			iStartInstID := iStartInstID +1;
			iStartLED := 	iStartLED +1;
			
			Q_sConvString:=	CONCAT(Q_sConvString,F_ToCHR(I_sStartZeichen));
			Q_sConvString:=	CONCAT(Q_sConvString,DINT_TO_STRING(I_diID));
			Q_sConvString:=	CONCAT(Q_sConvString,'.LED.');
			Q_sConvString:=	CONCAT(Q_sConvString,INT_TO_STRING(iStartInstID));
			Q_sConvString:=	CONCAT(Q_sConvString,'.ON.');
			Q_sConvString:=	CONCAT(Q_sConvString,INT_TO_STRING(I_iLED[iStartLED]));
			Q_sConvString:=	CONCAT(Q_sConvString,F_ToCHR(I_sEndZeichen));
		ELSE
			(* Externe LEDs*)
			iStartInstIDExt := 65;
			iStartLEDExt := 1;
			
			Q_sConvString:=	CONCAT(F_ToCHR(I_sStartZeichen),DINT_TO_STRING(I_diID));
			Q_sConvString:=	CONCAT(Q_sConvString,'.LED.');
			Q_sConvString:=	CONCAT(Q_sConvString,INT_TO_STRING(iStartInstIDExt));
			Q_sConvString:=	CONCAT(Q_sConvString,'.ON.');
			Q_sConvString:=	CONCAT(Q_sConvString,INT_TO_STRING(I_iLEDExt[iStartLEDExt]));
			Q_sConvString:=	CONCAT(Q_sConvString,F_ToCHR(I_sEndZeichen));
			
			iStartInstIDExt := iStartInstIDExt +1;
			iStartLEDExt := 	iStartLEDExt +1;
			
			Q_sConvString:=	CONCAT(Q_sConvString,F_ToCHR(I_sStartZeichen));
			Q_sConvString:=	CONCAT(Q_sConvString,DINT_TO_STRING(I_diID));
			Q_sConvString:=	CONCAT(Q_sConvString,'.LED.');
			Q_sConvString:=	CONCAT(Q_sConvString,INT_TO_STRING(iStartInstIDExt));
			Q_sConvString:=	CONCAT(Q_sConvString,'.ON.');
			Q_sConvString:=	CONCAT(Q_sConvString,INT_TO_STRING(I_iLEDExt[iStartLEDExt]));
			Q_sConvString:=	CONCAT(Q_sConvString,F_ToCHR(I_sEndZeichen));
			
			iStartInstIDExt := iStartInstIDExt +1;
			iStartLEDExt := 	iStartLEDExt +1;
			
			Q_sConvString:=	CONCAT(Q_sConvString,F_ToCHR(I_sStartZeichen));
			Q_sConvString:=	CONCAT(Q_sConvString,DINT_TO_STRING(I_diID));
			Q_sConvString:=	CONCAT(Q_sConvString,'.LED.');
			Q_sConvString:=	CONCAT(Q_sConvString,INT_TO_STRING(iStartInstIDExt));
			Q_sConvString:=	CONCAT(Q_sConvString,'.ON.');
			Q_sConvString:=	CONCAT(Q_sConvString,INT_TO_STRING(I_iLEDExt[iStartLEDExt]));
			Q_sConvString:=	CONCAT(Q_sConvString,F_ToCHR(I_sEndZeichen));
			
			iStartInstIDExt := iStartInstIDExt +1;
			iStartLEDExt := 	iStartLEDExt +1;
			
			Q_sConvString:=	CONCAT(Q_sConvString,F_ToCHR(I_sStartZeichen));
			Q_sConvString:=	CONCAT(Q_sConvString,DINT_TO_STRING(I_diID));
			Q_sConvString:=	CONCAT(Q_sConvString,'.LED.');
			Q_sConvString:=	CONCAT(Q_sConvString,INT_TO_STRING(iStartInstIDExt));
			Q_sConvString:=	CONCAT(Q_sConvString,'.ON.');
			Q_sConvString:=	CONCAT(Q_sConvString,INT_TO_STRING(I_iLEDExt[iStartLEDExt]));
			Q_sConvString:=	CONCAT(Q_sConvString,F_ToCHR(I_sEndZeichen));
			
			iStartInstIDExt := iStartInstIDExt +1;
			iStartLEDExt := 	iStartLEDExt +1;
			
			Q_sConvString:=	CONCAT(Q_sConvString,F_ToCHR(I_sStartZeichen));
			Q_sConvString:=	CONCAT(Q_sConvString,DINT_TO_STRING(I_diID));
			Q_sConvString:=	CONCAT(Q_sConvString,'.LED.');
			Q_sConvString:=	CONCAT(Q_sConvString,INT_TO_STRING(iStartInstIDExt));
			Q_sConvString:=	CONCAT(Q_sConvString,'.ON.');
			Q_sConvString:=	CONCAT(Q_sConvString,INT_TO_STRING(I_iLEDExt[iStartLEDExt]));
			Q_sConvString:=	CONCAT(Q_sConvString,F_ToCHR(I_sEndZeichen));
			
			iStartInstIDExt := iStartInstIDExt +1;
			iStartLEDExt := 	iStartLEDExt +1;
			
			Q_sConvString:=	CONCAT(Q_sConvString,F_ToCHR(I_sStartZeichen));
			Q_sConvString:=	CONCAT(Q_sConvString,DINT_TO_STRING(I_diID));
			Q_sConvString:=	CONCAT(Q_sConvString,'.LED.');
			Q_sConvString:=	CONCAT(Q_sConvString,INT_TO_STRING(iStartInstIDExt));
			Q_sConvString:=	CONCAT(Q_sConvString,'.ON.');
			Q_sConvString:=	CONCAT(Q_sConvString,INT_TO_STRING(I_iLEDExt[iStartLEDExt]));
			Q_sConvString:=	CONCAT(Q_sConvString,F_ToCHR(I_sEndZeichen));
		END_IF
	END_IF
ELSE
	(* Reset *)
	Q_sConvString:=	CONCAT(F_ToCHR(I_sStartZeichen),DINT_TO_STRING(I_diID));
	Q_sConvString:=	CONCAT(Q_sConvString,'.SYS.');
	Q_sConvString:=	CONCAT(Q_sConvString,INT_TO_STRING(1));
	Q_sConvString:=	CONCAT(Q_sConvString,'.RESET');
	Q_sConvString:=	CONCAT(Q_sConvString,F_ToCHR(I_sEndZeichen));
END_IF

END_FUNCTION_BLOCK

// ---- POUs/RS485_Hausbus_FB/RS485 COM/fb_RS485Ping.TcPOU
(*======================================================================================================================================*)
(*fb_RS485Ping:	Einfacher Universal Ping Baustein um von allerlei Geräten von haus-bus.de Kommunikation zu Checken über RS485 
				im gegensatz zum ComCheck Baustein wird hier nur gelesen, da es Geräte gibt, welche entweder Zyklich selbst 
				ein Lebenszeichen geben z.B. CYD oder die 6Fach Taster (Helligkeit, Temp, Luftfeuchtigkeit).
				Besonderheit bei dem 6Fach Taster ist: nach einem Reset werden immer auch StatusTelegramme gesendet. 
				Damit lässt sich dann auch festellen ob ein Taster Online ist. 
				Für die Aktoren ist dieser Baustein eher weniger geeignet, da es dort keine Zyklischen Telegramme gibt und 
				auch nach einem Reset keine Statustelegramme gesendet werden! 
				
				Der Baustein kann auch verwendet werden um einfach nur zu überwachen, ob ein Teilnehmer noch online ist über langen
				Zeitraum- Dafür muss der Timeout einfach sehr Hoch gestellt werden - z.B 120 Minuten und bAutoPing Aktiviert sein 
			
				Wenn I_bAutoPing nicht Aktiv ist, wird nur eine Ping überprüfung beim Aktivieren des Bausteins über I_bExecute 
				durchgeführt. Wenn die Prüfung erfolgreich ist, wird der Status Q_bComOk gesetzt. Der Status Q_bComOk wird erst durch 
				I_bReset wieder zurück gesetzt. 
				
				Wenn I_bAutoPing Aktiv ist, wird sobald der Baustein über I_bExecute gestartet wurde, und ein Ping Aufgebaut ist, 
				immer nach ablauf der Zeit: I_tPingTimeout erneut der Ping geprüft. Sollte der Ping nicht kommen, so wird nach ablauf der 
+				Zeit: I_tPingTimeout in den Timepout gesprungen. Dann kann nur über einen Reset durch: I_bReset erneut gestartet werden*)
(*
Date          	| Version    	| created under        	| Author          	| Remark *)
(*====================================================================================================================================================*)
(*27/05/2025   	| 1.00      		| TC3		  		| N.Kersting       | first release *)
(*====================================================================================================================================================*)
FUNCTION_BLOCK fb_RS485Ping
VAR_INPUT
	I_bExecute			:BOOL;							(* Aktiviert den Ablauf *)
	I_bAutoPing			:BOOL;							(* Aktiviert die Automatische Prüfung, wenn aus- wird nur einmal beim Aktivieren über bExecute geprüft *)
	I_bAutoReset		:BOOL;							(* Aktiviert das Automatische wieder Quittieren wenn der Ping nicht empfangen wurde *)
	I_bReset			:BOOL;							(* Setzet den Ping und die Ablauf zurück *)
	I_tPingTimeout		:TIME := T#2S;					(* Zeit, bis der Ping gekommen sein muss *)
	I_diID				:DINT;							(* Device ID *)
	I_sStartZeichen		:BYTE := 16#FD;					(* Startzeichen Präfix *)
	I_sEndZeichen		:BYTE := 16#FE;					(* Endzeichen Suffix *)
	I_StringReceived	:STRING(255);					(* Empfangener String *)
END_VAR
VAR_OUTPUT		
	Q_sState			:STRING;						(* Status  *)
	Q_bComOk			:BOOL;							(* Verbindung Aufgebaut *)
	Q_bTimeout			:BOOL;							(* Timeout  *)
END_VAR
VAR
	bResetCnt			:BOOL;
	tonTimeout			:ton;
	icntSymbole			:INT;
	iStep				:INT;
	i					:INT;
	fbBusPingEvent		:fb_BusPingEvent;
	bCOMMem				:BOOL;
	rTrigFailCount		:r_trig;
	
	dwCntFail			:DWORD;
END_VAR

(* Timeout Zeit *)
tonTimeout(
	PT:= I_tPingTimeout);

(* Ping Fehler Zählen *)	
rTrigFailCount();
	
(* Reset ausführen *)
IF I_bReset 
	OR NOT I_bExecute
THEN
	iStep := 0;	
END_IF

(* Timeout Counter auf 0 Setzen *)
IF bResetCnt
THEN
	dwCntFail := 0;
END_IF
	
(* Ablauf *)
CASE iStep OF
(*=========================================================*)	
0:	Q_sState := 'INIT';
	Q_bComOk := FALSE;
	bCOMMem := FALSE; (* Ping zurück setzen *)
	tonTimeout.IN := FALSE;
	Q_bTimeout := FALSE;
	rTrigFailCount.CLK := FALSE;
	
	IF I_bExecute
	THEN
		iStep := iStep +1;
	END_IF
	
(*=========================================================*)	
1:	Q_sState :=  'Warten auf Ping ';	
	tonTimeout.IN := TRUE;
	
	IF fbBusPingEvent.Q_bOut
	THEN
		tonTimeout.IN := FALSE;
		bCOMMem := TRUE;
		iStep := 998;
	ELSIF
		tonTimeout.Q
	THEN
		tonTimeout.IN := FALSE;
		Q_bTimeout := TRUE;
		Q_bComOk := FALSE;
		Q_sState :=  'Timeout- Kein Ping empfangen';	
		iStep := -1;
	END_IF

(*=========================================================*)	
998: Q_sState :=  'Ping empfangen, Warte das String Leer ist';	
	tonTimeout.IN := TRUE;
	
	IF NOT fbBusPingEvent.Q_bOut
	THEN
		iStep := 999;
	ELSIF
		tonTimeout.Q
	THEN
		tonTimeout.IN := FALSE;
		Q_bTimeout := TRUE;
		Q_bComOk := FALSE;
		Q_sState :=  'Timeout String wurde nicht geleert!';	
		iStep := -998;
	END_IF
	
(*=========================================================*)	
999: Q_sState :=  'Ping empfangen, erfolgreich Verbunden!';		
	Q_bComOk := TRUE;
	Q_bTimeout := FALSE;
	
	(* Die Verbindung wurde nun geprüft, kann aber nur über
		I_bReset wieder erneut geprüft werden ! *)
	
	IF I_bAutoPing
	THEN
		tonTimeout.IN := TRUE;
		
		IF tonTimeout.Q
		THEN
			tonTimeout.IN := FALSE;
				
			IF I_bExecute
			THEN
				iStep := 1;	(* Erneut Prüfen *)
			END_IF
		END_IF
	ELSE
		tonTimeout.IN := FALSE;
	END_IF
ELSE
(*=========================================================*)	
(*	Timeout *)	
	rTrigFailCount.CLK := TRUE;
	
	IF rTrigFailCount.Q
	THEN
		dwCntFail := dwCntFail+1;
	END_IF
	(*	Automatische Quittierung *)	
	IF 	I_bAutoReset
	THEN
		tonTimeout.IN := TRUE;
		
		IF tonTimeout.Q
			OR fbBusPingEvent.Q_bOut
		THEN
			tonTimeout.IN := FALSE;
			
			IF I_bExecute
			THEN
				rTrigFailCount.CLK := FALSE;
				iStep := 1;	(* Erneut Prüfen *)
			END_IF
		END_IF
	END_IF
END_CASE


(* Durchgehend Checken ob Ping kommt *)
fbBusPingEvent(
	I_bReset := 			FALSE,
	I_sID:= 				DINT_TO_STRING(I_diID ), 
	I_sReceivedString:= 	I_StringReceived, 
	Q_bOut=> 				);

END_FUNCTION_BLOCK

// ---- POUs/RS485_Hausbus_FB/RelaisModul/fb_RelaisBus16F.TcPOU
(*======================================================================================================================================*)
(*fb_RelaisBus16F:		Einfache RS485 Kommunikation für Haus-bus.de Komponenten zum testen 	
						 *)
(*
Date          	| Version    	| created under        	| Author          	| Remark *)
(*====================================================================================================================================================*)
(*08/05/2025   	| 1.00      		| TC3		  		| N.Kersting       	| first release *)
(*08/05/2025   	| 1.01      		| TC3		  		| N.Kersting       	| Relais in Sections aufgeteilt um String Länge zu verringern *)
(*09/05/2025   	| 1.02      		| TC3		  		| N.Kersting       	| Ping Versuche Implementiert mit Globalen Parametern *)
(*10/05/2025   	| 2.00      		| TC3		  		| N.Kersting      	| Umstellung auf Externe FiFo Sendebaustein *)
(*12/05/2025   	| 2.01      		| TC3		  		| N.Kersting      	| Verriegelung für ComCheck hinzugefügt und Relais Sections auf 2 redzuziert *)
(*13/05/2025   	| 3.00      		| TC3		  		| N.Kersting       	| Viele Bugs gefixt, bei Änderung der Ausgängen wird nun eine Anforderung gesetzt  *)
(*28/05/2025   	| 3.01      		| TC3		  		| N.Kersting        | Neuen Einfachen Ping Baustein, welcher nicht sendet, nur auswertet implementiert *)
(*====================================================================================================================================================*)
FUNCTION_BLOCK fb_RelaisBus16F
VAR_INPUT
	I_FifoID			:INT;
	I_bPingStart		:BOOL;						(* Ping Done vom Vorheriegen*)
	I_stInput			:ST_BusRelais16F_Input;
	I_StringReceived	:STRING(255);
END_VAR
VAR_OUTPUT
	Q_sFiFoSend			:STRING(255);
   	Q_stOutput			:ST_BusRelais16F_Output;
	Q_stCnt				:ST_BusRelais16F_Cnt;
END_VAR
VAR
(*----------------------------------------------*)
(* Interne Parameter*)
(*----------------------------------------------*)		
	bSetExecute			:BOOL := TRUE;				(* Aktiviert die Schrittketten, welche Telegramme versenden *)
	bCheckPing			:BOOL := TRUE;				(* Ping Checken Schrittkette Aktivieren *)
	sStartZeichen		:BYTE := 16#FD;				(* Startzeichen Präfix *)
	sEndZeichen			:BYTE := 16#FE;				(* Endzeichen Suffix *)
	iAnzResetSend		:INT := 2;					(* Anzahl der Sendeversuche bei Reset *)
	tPingTimer			:TIME:= T#5S;				(* Zeit, bis wiederholend der Ping versendet wird *)
	tReceiveTimeout		:TIME:= T#2S;				(* Zeit, bis die Event Schrittkette für das Empfangen Automatisch neu Startet*)
	tStartupLEDOn		:TIME:= T#3S;				(* Zeit, wie Lange die LEDS beim Startup kurz eingeschaltet werden *)
	tResetTimeout		:TIME:= T#8S;				(* Zeit, bis bei einem Reset es zu einem Fehler kommt, wenn kein Ping empfangen wird *)
	tResetReboot		:TIME:= T#3S;				(* Zeit, die nach einem Reset Abgewaretet wird damit das Gerät neustarten kann*)
	tResetStartup		:TIME:= T#1S;				(* Zeit, die nach einem Reset Abgewaretet wird bis ein Startup ausgeführt wird nach dem erhalt des Pings vom Gerät*)
	tStartupAfterReset	:TIME := T#5S;				(* Zeit, wann das Startup Zurückgesetzt wird, wenn der Ping verloren wird *)
(*----------------------------------------------*)
(* Strings *)
(*----------------------------------------------*)			
	sSendString			:STRING(255);
	sFiFoSend			:STRING(255);
	sReceived			:STRING(255);
	sLastSendString		:STRING(255);
	sLastSendString1	:STRING(255);
	sStateReset			:STRING;
(*----------------------------------------------*)
(* Funktionsbausteine *)
(*----------------------------------------------*)
	fbBusTasterEvent	:ARRAY[1..8] OF fb_BusTasterEvent;		(* Interne 8 Taster Abfragen *)
	fbStringConvR1B6F	:fb_StringConvRB16F;
	fbPing				:fb_RS485Ping;
(*----------------------------------------------*)
(* Indexe *)
(*----------------------------------------------*)	
	iDeviceStartup		:INT :=0;	(* Startup Schrittkette *)
	sDeviceStartup		:STRING;
    iState     			:INT := 0;
	iStepSet			:INT;
	i,h,j,l				:INT;
	idxLED				:INT;
	idxBtn				:INT := 1;
	ibOutMem			:ARRAY[1..16] OF BOOL;
	ibOutAnf			:ARRAY[1..16] OF BOOL;
	cntChangesOut		:INT;
	icntResetSend		:INT;
	iSection			:INT :=1;
	iMaxPingTry			:INT := 5;
(*----------------------------------------------*)
(* Timer/Trigger *)
(*----------------------------------------------*)		
	r_trigStartupAfterReset	:r_trig;
	r_TrigReset				:r_trig;		
	r_TrigCountBtn			:ARRAY[1..16] OF r_trig;
	
	tonStartupAfterReset	:ton;
	tonReceiveTimeout		:ton;
	tonResetTimeout			:ton;
	tonResetDone			:ton;
	tonStepStartup			:ton;
(*----------------------------------------------*)
(* Status *)
(*----------------------------------------------*)			
	bPingOK					:BOOL;
	bErrorEvent				:BOOL;
	bErrorPing				:BOOL;
	bErrorSet				:BOOL;
	bErrorReset				:BOOL;
	bResetBusy				:BOOL;
	bResetDone				:BOOL;
	bResetAutoStart			:BOOL;
	bStartupStart			:BOOL;
	bStartupDone			:BOOL;	
	bMemExt					:BOOL;
	bStartUpCheckPing		:BOOL;
	bActivateSend			:BOOL;
	bReadyToPing			:BOOL;
	bSendeAnforderung		:BOOL;
END_VAR

(*============================================================================================*)
(* Parameter *)
tPingTimer :=		GVL_HausBus_Parameter.cTimePingTimeRelais;
tReceiveTimeout :=	GVL_HausBus_Parameter.cTimeReceiveTimeoutRelais;
bCheckPing :=		GVL_HausBus_Parameter.bUseRelaisPing;
iMaxPingTry :=		GVL_HausBus_Parameter.cMaxPingTry;

(*============================================================================================*)
(* Startup Zurücksetzen Reset *)
r_TrigReset(CLK := I_stInput.bReset);

(* Startup Zurücksetzen bei Busverlust *)
tonStartupAfterReset(
	IN := NOT bPingOK
			AND bCheckPing,
	PT:= tStartupAfterReset);

r_trigStartupAfterReset
	(CLK := tonStartupAfterReset.Q);
	
IF NOT I_stInput.bExecute
	OR r_TrigReset.Q
	OR r_trigStartupAfterReset.Q
THEN
	iDeviceStartup := 0;
END_IF

(*============================================================================================*)
(* Ping Dauerhaft Senden*)
ac02_Ping();
	
(*============================================================================================*)
(* Startup Schrittkette *)
CASE iDeviceStartup OF
(*============================================================================================*)
0: 	sDeviceStartup := 'INIT';
	bResetDone := FALSE;
	bStartupDone := FALSE;
	bStartupStart := FALSE;
	bResetAutoStart := FALSE;
	bStartUpCheckPing := FALSE;
	bActivateSend := FALSE;
	bReadyToPing := TRUE;
	
	iStepSet := 0;
	
	IF 	I_stInput.bExecute
	THEN
		iDeviceStartup := iDeviceStartup+1;
	END_IF
(*============================================================================================*)
1: 	sDeviceStartup := 'Device ID Prüfen';
	
	IF  I_stInput.diID <> 0
	THEN
		iDeviceStartup := iDeviceStartup+1;
	ELSE
		sDeviceStartup := 'ERROR- Device ID Prüfen';
	END_IF
(*============================================================================================*)
2: 	sDeviceStartup := 'Verbindung Prüfen';
	bActivateSend := TRUE;	(* Senden Aktivieren *)
	iDeviceStartup := iDeviceStartup+1;
	(*
	sDeviceStartup := CONCAT(sDeviceStartup,fbRS485ComCheck.Q_sState);
	
	IF fbRS485ComCheck.Q_bComOk
		OR NOT bCheckPing
	THEN
		iDeviceStartup := iDeviceStartup+1;
	END_IF*)

(*============================================================================================*)
3: 	sDeviceStartup := 'Reset Ausführen';	
	bActivateSend := TRUE;	(* Senden Aktivieren *)
	
	(*	RESET Device *)
	ac01_SetReset();
	bResetAutoStart := TRUE;
	
	sDeviceStartup :=	CONCAT(sDeviceStartup,sStateReset);
	
	IF bResetDone
	THEN
		iStepSet := 0;
		iDeviceStartup := iDeviceStartup+1;
	END_IF

(*============================================================================================*)
4: 	sDeviceStartup := 'Startup Ausführen';
		
	(* LED Setzen *)
	ac01_SetOutput();
	
	bStartupStart := TRUE;
	
	IF bStartupDone 
	THEN
		bStartupStart := FALSE;
		iDeviceStartup := 999;
	END_IF

(*============================================================================================*)
999: 
	(*bReadyToPing := NOT fbRS485SendCmd.Q_bBusy;*)
	
	(* LED Setzen *)
	ac01_SetOutput();
	
	(* Events Auslesen *)
	ac00_Event();
	
	(* Zähler *)
	ac10_Counter();
	
	sDeviceStartup := 'Startup Ausgeführt- Gerät im OP';
	
END_CASE

(*============================================================================================*)
(* Sendebaustein *)
IF bActivateSend
THEN
	Q_sFiFoSend :=	sFiFoSend;
END_IF

(*============================================================================================*)	
(* Zähler *)
ac10_Counter();
	
(*============================================================================================*)
(* Outputs *)
Q_stOutput.bCOM :=		bPingOK;

Q_stOutput.bError := 	bErrorEvent
						OR bErrorPing
						OR bErrorSet
						OR (NOT bPingOK
						AND bCheckPing);
						
Q_stOutput.bStartupDone	:=	bStartupDone;

Q_stOutput.sState :=	CONCAT(I_stInput.sName,'| ');
Q_stOutput.sState :=	CONCAT(Q_stOutput.sState, sDeviceStartup);

ACTION ac00_Event:
(*============================================================================================*)
(*	EVENT Schrittkette *)
(*============================================================================================*)
sReceived := I_StringReceived;
	
FOR i := 1 TO 8 BY 1 DO 
	fbBusTasterEvent[i](
		I_sID:= 				DINT_TO_STRING(I_stInput.diID), 
		I_sInstID:= 			INT_TO_STRING(i+96), 
		I_sReceivedString:= 	sReceived, 
		Q_bOut=> 				Q_stOutput.bInputs[i]);
END_FOR
END_ACTION

ACTION ac01_SetOutput:
(*============================================================================================*)
(*	LED Helligkeit Setzen/ Startup Schrittkette *)
(*============================================================================================*)

(* Einfaches Setzen der LED Helligkeiten (0-100 Prozent *)
(* Neu, es werden alle LEDs zu einem String zusammengefügt und Gleichzeitig gesetzt *)
tonStepStartup(
	PT:= tStartupLEDOn);

cntChangesOut := 0;
FOR l := 1 TO 16 BY 1 DO
	IF ibOutMem[l] <> I_stInput.bOut[l]
	THEN
		cntChangesOut := cntChangesOut +1;
	END_IF
END_FOR
	
CASE iStepSet OF
(*============================================================================================*)
0:	(* INIT und warten auf Change *)
	tonStepStartup.IN := FALSE;
	iSection := 1;
	
	(* Merken ob eine Anforderung Ansteht *)
	IF cntChangesOut <>0
	THEN
		bSendeAnforderung := TRUE;
		FOR h := 1 TO 16 BY 1 DO
			ibOutAnf[h] := I_stInput.bOut[h];
		END_FOR
	END_IF
	
	IF (bSendeAnforderung
		AND bSetExecute)
		AND NOT bStartupStart
	THEN
		bSendeAnforderung := FALSE;
		(* Angeforderten Relaiszustand speichern *)
		FOR h := 1 TO 16 BY 1 DO
			ibOutMem[h] := I_stInput.bOut[h];
		END_FOR
		iStepSet := 10;
	ELSIF
		bStartupStart
	THEN
		iStepSet := 100;	(* Startup *)
	END_IF
	
(*============================================================================================*)
10:	(* String senden *)	
	(* Nur Relais Schreiben *)
	
	fbStringConvR1B6F(
		I_bReset:= 			FALSE, 
		I_bRedLEDOn:= 		FALSE, 
		I_bRedLEDOff:= 		FALSE, 
		I_iSection :=		iSection,
		I_diID:= 			I_stInput.diID, 
		I_bOut:= 			ibOutAnf, 
		I_sStartZeichen:= 	sStartZeichen, 
		I_sEndZeichen:= 	sEndZeichen,	 
		Q_sConvString=> 	sSendString);
		
	(* Senden an FiFo*)
	IF GVL_RS485FiFoSend.bSendDoneFiFo[I_FifoID]
	THEN
		sFiFoSend :=	sSendString;
	END_IF
	IF NOT GVL_RS485FiFoSend.bSendDoneFiFo[I_FifoID]
	THEN
		IF iSection <= 2
		THEN
			iSection :=	iSection+1;
		END_IF
		
		iStepSet := 20;
	END_IF
		
(*============================================================================================*)	
20:	(* Warten bis nicht Busy *)	
	IF GVL_RS485FiFoSend.bSendDoneFiFo[I_FifoID]	
	THEN
		sFiFoSend := ''; 
		
		IF iSection <= 2
		THEN
			sLastSendString :=	sSendString;
			iStepSet := 10;
		ELSE
			sLastSendString1 :=	sSendString;
			iStepSet := 0;
		END_IF
	END_IF
	
(*============================================================================================*)	
(* Startup  *)
100:	tonStepStartup.IN := TRUE;
	
	IF tonStepStartup.Q
	THEN
		iStepSet := 110;
	END_IF
	
(*============================================================================================*)
110:(* String senden *)	(* Alle Relais Ausschalten *)
	tonStepStartup.IN := FALSE;
		
	fbStringConvR1B6F(
		I_bReset:= 			FALSE, 
		I_bRedLEDOn:= 		FALSE, 
		I_bRedLEDOff:= 		FALSE, 
		I_iSection :=		iSection,
		I_diID:= 			I_stInput.diID, 
		I_bOut:= 			I_stInput.bOut, 
		I_sStartZeichen:= 	sStartZeichen, 
		I_sEndZeichen:= 	sEndZeichen,	 
		Q_sConvString=> 	sSendString);
		
	IF GVL_RS485FiFoSend.bSendDoneFiFo[I_FifoID]
	THEN
		sFiFoSend :=	sSendString;
	END_IF
	IF NOT GVL_RS485FiFoSend.bSendDoneFiFo[I_FifoID]
	THEN
		IF iSection <= 2
		THEN
			iSection :=	iSection+1;
		END_IF
		
		iStepSet := 111;
	END_IF
	
(*============================================================================================*)
111:(* String senden *)
	IF GVL_RS485FiFoSend.bSendDoneFiFo[I_FifoID]
	THEN
		sLastSendString :=	sSendString;
		sFiFoSend := ''; 
		
		IF iSection <= 2
		THEN
			iStepSet := 110;
		ELSE
			iStepSet := 112;
		END_IF
	END_IF
	
(*============================================================================================*)
112:(* String senden *)	(* Rote LED Einschalten *)
	tonStepStartup.IN := FALSE;
		
	fbStringConvR1B6F(
		I_bReset:= 			FALSE, 
		I_bRedLEDOn:= 		TRUE, 
		I_bRedLEDOff:= 		FALSE, 
		I_diID:= 			I_stInput.diID, 
		I_bOut:= 			I_stInput.bOut, 
		I_sStartZeichen:= 	sStartZeichen, 
		I_sEndZeichen:= 	sEndZeichen,	 
		Q_sConvString=> 	sSendString);
					
	IF GVL_RS485FiFoSend.bSendDoneFiFo[I_FifoID]
	THEN
		sFiFoSend :=	sSendString;
	END_IF
	IF NOT GVL_RS485FiFoSend.bSendDoneFiFo[I_FifoID]
	THEN
		iStepSet := 113;
	END_IF
	
(*============================================================================================*)
113:(* String senden *) (* Warten *)
	IF GVL_RS485FiFoSend.bSendDoneFiFo[I_FifoID]
	THEN
		sFiFoSend := ''; 
		tonStepStartup.IN := TRUE;
		
		IF tonStepStartup.Q
		THEN
			tonStepStartup.IN := FALSE;
			iStepSet := 114;
		END_IF
	END_IF

(*============================================================================================*)
114:(* String senden *)	(* Rote LED Ausschalten *)
	tonStepStartup.IN := FALSE;
	
	fbStringConvR1B6F(
		I_bReset:= 			FALSE, 
		I_bRedLEDOn:= 		FALSE, 
		I_bRedLEDOff:= 		TRUE, 
		I_diID:= 			I_stInput.diID, 
		I_bOut:= 			I_stInput.bOut, 
		I_sStartZeichen:= 	sStartZeichen, 
		I_sEndZeichen:= 	sEndZeichen,	 
		Q_sConvString=> 	sSendString);
			
	IF GVL_RS485FiFoSend.bSendDoneFiFo[I_FifoID]
	THEN
		sFiFoSend :=	sSendString;
	END_IF
	IF NOT GVL_RS485FiFoSend.bSendDoneFiFo[I_FifoID]
	THEN
		iStepSet := 120;
	END_IF
	
(*============================================================================================*)	
120:(* Warten bis nicht Busy *)	
	IF GVL_RS485FiFoSend.bSendDoneFiFo[I_FifoID]
	THEN
		sFiFoSend := ''; 
				
		tonStepStartup.IN := TRUE;
	
		IF tonStepStartup.Q
		THEN
			bStartupDone := TRUE;
			tonStepStartup.IN := FALSE;
			bStartupStart := FALSE;
			iStepSet := 10;	(* Anschließend noch einmal die Eingangs Helligkeit setzen *)
		END_IF
	END_IF	

END_CASE
END_ACTION

ACTION ac01_SetReset:
(*============================================================================================*)
(*	RESET Schrittkette *)
(*============================================================================================*)
tonResetTimeout(
	PT := tResetTimeout);

tonResetDone();

(* Einfaches Setzen der LED Helligkeiten (0-100 Prozent *)
CASE iStepSet OF
(*============================================================================================*)
0:	sStateReset := 'INIT';
	
	IF (bSetExecute
		AND (I_stInput.bReset
		OR bResetAutoStart))
	THEN
		bStartupDone := FALSE;
		bResetDone := FALSE;
		tonResetTimeout.IN := FALSE;
		tonResetDone.IN := FALSE;
		icntResetSend := 0;
		
		(* Ausgänge alle auf 0 setzen *)
		FOR h := 1 TO 16 BY 1 DO
			ibOutMem[h] := FALSE;
			Q_stOutput.bInputs[h] := FALSE;
		END_FOR
		
		bPingOK := FALSE;
		
		iStepSet := iStepSet +1;
	END_IF

(*============================================================================================*)	
1:	sStateReset := 'Sende Reset Befehl';
	bResetBusy := TRUE;
	bErrorReset := FALSE;
	
	fbStringConvR1B6F(
		I_bReset:= 			TRUE, 
		I_bRedLEDOn:= 		FALSE, 
		I_bRedLEDOff:= 		FALSE, 
		I_diID:= 			I_stInput.diID, 
		I_bOut:= 			I_stInput.bOut, 
		I_sStartZeichen:= 	sStartZeichen, 
		I_sEndZeichen:= 	sEndZeichen,	 
		Q_sConvString=> 	sSendString);

	(* Senden an FiFo*)
	IF GVL_RS485FiFoSend.bSendDoneFiFo[I_FifoID]
	THEN
		sFiFoSend :=	sSendString;
	END_IF
	IF NOT GVL_RS485FiFoSend.bSendDoneFiFo[I_FifoID]
	THEN
		iStepSet := iStepSet+1;
	END_IF

(*============================================================================================*)
2:	sStateReset := 'Sende Reset Befehl';

	IF GVL_RS485FiFoSend.bSendDoneFiFo[I_FifoID]
	THEN
		sFiFoSend := ''; 
		
		fbStringConvR1B6F(
			I_bReset :=			FALSE);
		iStepSet := 3;
	END_IF
	
(*============================================================================================*)	
3:	sStateReset := 'Reset durchgeführt, Warte auf Ping';
	tonResetDone.IN := TRUE;
	tonResetDone.PT := tResetReboot;
		
	iState := 0;
	
	IF tonResetDone.Q
	THEN
		tonResetDone.IN := FALSE;
		iStepSet := 4;
	END_IF
	
(*============================================================================================*)	
4:	sStateReset := 'Warte auf Ping vom Gerät';	
	tonResetTimeout.IN := TRUE;
	bStartUpCheckPing := TRUE;
	
	IF bPingOK 
	THEN
		bErrorReset := FALSE;
		tonResetTimeout.IN := FALSE;
		iStepSet := 5;
	ELSIF
		tonResetTimeout.Q
	THEN
		sStateReset := 'Ping Timeout, keine Kommunikation';
		bErrorReset := TRUE;

		IF I_stInput.bReset
		THEN
			bResetBusy := FALSE;
			iStepSet := 0;
		END_IF
	END_IF

(*============================================================================================*)
5:	sStateReset := 'Startup Aktiv';
	
	tonResetDone.IN := NOT I_stInput.bReset;
	tonResetDone.PT := tResetStartup;

	sFiFoSend := ''; 
	
	IF tonResetDone.Q
	THEN
		fbStringConvR1B6F(
			I_bReset :=			FALSE);
			
		sStateReset := 'Ping erhalten, Reset Erfolgreich';
		bResetAutoStart := FALSE;
		bResetDone := TRUE;
		bResetBusy := FALSE;
		iState := 0;
		iStepSet := 0;
	END_IF
END_CASE
END_ACTION

ACTION ac02_Ping:
(*============================================================================================*)
(* 	Ping Bautsein, Checkt ob die Kommunikation vorhanden ist *)
(*============================================================================================*)
fbPing(
	I_bExecute:= 			bStartUpCheckPing, 
	I_bAutoPing:= 			bCheckPing, 
	I_bAutoReset:= 			bCheckPing, 
	I_bReset:= 				r_TrigReset.Q
							OR NOT bStartUpCheckPing, 
	I_tPingTimeout:= 		tPingTimer, 
	I_diID:= 				I_stInput.diID, 
	I_sStartZeichen:= 		sStartZeichen, 
	I_sEndZeichen:= 		sEndZeichen, 
	I_StringReceived:= 		I_StringReceived, 
	Q_sState=> , 
	Q_bComOk=> 				bPingOK, 
	Q_bTimeout=> 			bErrorPing);
END_ACTION

ACTION ac10_Counter:
(*============================================================================================*)
(* 	Zähler *)
(*============================================================================================*)
FOR j := 1 TO 16 BY 1 DO 
	r_TrigCountBtn[j](
		CLK := I_stInput.bOut[j]);
		
	IF r_TrigCountBtn[j].Q
	THEN
		Q_stCnt.dwCntRelais[j] := Q_stCnt.dwCntRelais[j]+1;
	END_IF
	
END_FOR
END_ACTION

ACTION ac99_Doku:
(*======================================================================================================================================*)
(*	DOKU	*)
(*======================================================================================================================================*)
(* Wichtiger Hinweis:
		-Bei dem 6 Fach Taster ist zu Beachten, dass es nur 4 Externe EA/s gibt also 4 LEDs und 4 Taster, 
		da der ESP 32 Nur 10Es und 10As besitzt.
		- Die 4 Zusätzlichen Ausgänge werden von der Hintergrundbeleuchtung Ausgeschlossen und müssen über den Befehl: SET_MBR einzeln 
			gesetzt werden! *)	
	
(* Verdrahtung:		
	Verdrahtung füR: KL6041
        +-------+
        |       |
        | TxD+ ----+
        |         |----> RS485 A (zum Bus)
        | RxD+ ----+
        |         |
        | TxD− ----+
        |         |----> RS485 B (zum Bus)
        | RxD− ----+
        +-------+	*)
		
(*======================================================================================================================================*)
(* Telegrammbeschreibung *)

(*	Die XML Dateien der verschiedenen Module sind grundsätzlich immer gleich aufgebaut. 
	Je Instanz der verschiedenen Sensoren und Aktoren werden die zu sendenden Befehle bzw. 
	die zu empfangenen Events beschrieben. 
	Alle Telegramme sind ASCII kodiert und sind umgeben mit dem binären Startzeichen 0xFD und dem binären Endezeichen 0xFE.

	Grundaufbauer aller im Folgenden beschriebenen Telegramme:
	
	-Startzeichen immer 0xFD.
	-Punkte dienen als Trennzeichen der verschiedenen Elemente
	-Endezeichen immer 0xFE.
	-Element 1 ist die Geräte-ID, die entsprechend der verwendeten Module angepasst werden muss (hier beispielhaft jeweils 12345)
	-Element 2 ist ein Schlüsselwort für den jeweiligen Funktionstyp (z.b. BTN, LED, DIM, usw)
	-Element 3 ist die InstanzID gemäß XML Templates (also welche Taster oder welcher Dimmer konkret gemeint ist)
	-Element 4 zeigt die jeweilige Aktion zum Funktionstypen (z.b. ON, OFF, STATUS)
	-Anschließend kommen optional diverse Parameter, die mit P1,P2,...P3 bezeichnet werden
	
	Im Folgenden wird nur noch auf die speziellen Telegramdaten eingegangen:
	
	(*------------------------------------------------------------*)
	Taster oder digitaler Eingang (Sensor):
	(*------------------------------------------------------------*)
	Telegram Event:  	
	
	\xFD 12345.BTN.17.STATUS.P1 \xFE
	
		Funktionstyp:		BTN (kurz für Button)
		Instanz-ID:			hier 17 (in XML nachschauen)
		Aktion:				STATUS
		P1:					1, wenn Taste gedrückt bzw. Eingang aktiv
							0, wenn Taste losgelassen bzw. Eingang inaktiv
	
	Telegram Statusabfrage:  	
	
	\xFD 12345.BTN.17.gSTATUS \xFE
	
		Antwort:  			\xFD 12345.BTN.17.rSTATUS.P1 \xFE
		P1:					1, wenn Taste gedrückt bzw. Eingang aktiv
							0, wenn Taste losgelassen bzw. Eingang inaktiv

	(*------------------------------------------------------------*)
	Led (Aktor):
	(*------------------------------------------------------------*)
	Telegram Helligkeit setzen:  	
	
	\xFD 12345.LED.50.ON.P1.P2.P3 \xFE
	
		Funktionstyp:			LED
		Instanz-ID:				hier 50 (in XML nachschauen)
		Aktion:					ON
		P1:						gewünschte Helligkeit 0-100
		P2:						Einschaltdauer in 100stel Sekunden (0 = daueran)
		P3:						Einschaltverzögerung in Sekunden (0 = ohne Verzögerung)
	
	Telegram Mindesthelligkeit:  	
	
	\xFD 12345.LED.50.SET_MBR.P1 \xFE
		
		Aktion:					SET_MBR (Setzt eine Mindesthelligkeit, die auch dann erhalten bleibt, wenn man per OFF ausschaltet)
		P1:						gewünschte Helligkeit 0-100
	
	Telegram Statusabfrage:  	

	\xFD 12345.LED.50.gSTATUS \xFE
	
		Antwort:  				\xFD 12345.LED.50.rSTATUS.P1.P2 \xFE
		P1:						aktuelle Helligkeit 0-100
		P2:						Einschaltdauer in 100stel Sekunden
	
	(*------------------------------------------------------------*)
	Hintergrundbeleuchtung (Aktor):
	(*------------------------------------------------------------*)
	Telegram Minhelligkeit:  
	
	\xFD 12345.LBN.16.SET_MBR.P1 \xFE
	
		Aktion:					SET_MBR ((Setzt eine Mindesthelligkeit, die auch dann erhalten bleibt, wenn man per OFF ausschaltet)
		P1:						gewünschte Helligkeit 0-100
		
	Telegram Statusabfrage:  	

	\xFD 12345.LBN.16.gSTATUS \xFE
	
		Antwort:  				\xFD 12345.LBN.16.rSTATUS.P1 \xFE
		P1:						aktuelle Helligkeit 0-100

	(*------------------------------------------------------------*)
	Temperatursensor (Sensor):
	(*------------------------------------------------------------*)
	Telegram Event:  	
	
	\xFD 12345.TMP.1.STATUS.P1.P2 \xFE
	
		Funktionstyp:			TMP (kurz für Temperatur)
		Instanz-ID:				hier 1 (in XML nachschauen)
		Aktion:					STATUS
		P1:						Temperatur in Grad Vorkommastellen
		P2:						Temperatur in Grad Nachkommastellen
	
	Telegram Statusabfrage:  
	
	\xFD 12345.TMP.1.gSTATUS \xFE
	
		Antwort:  				\xFD 12345.TMP.1.rSTATUS.P1.P2 \xFE
		P1:						Temperatur in Grad Vorkommastellen
		P2:						Temperatur in Grad Nachkommastellen

	(*------------------------------------------------------------*)
	Feuchtesensor (Sensor):
	(*------------------------------------------------------------*)
	Telegram Event:  	

	\xFD 12345.RHD.1.STATUS.P1.P2 \xFE
	
		Funktionstyp:			RHD (kurz für Relative Humidity)
		Instanz-ID:				hier 1 (in XML nachschauen)
		Aktion:					STATUS
		P1:						Relative Luftfeuchtigkeit 0-100 Vorkommastellen
		P2:						Relative Luftfeuchtigkeit 0-100 Nachkommastellen

	Telegram Statusabfrage:  	
	
	\xFD 12345.RHD.1.gSTATUS \xFE
	
	Antwort:  					\xFD 12345.RHD.1.rSTATUS.P1 \xFE
	P1:							Relative Luftfeuchtigkeit 0-100 Vorkommastellen
	P2:							Relative Luftfeuchtigkeit 0-100 Nachkommastellen

	(*------------------------------------------------------------*)
	Helligkeitssensor (Sensor):
	(*------------------------------------------------------------*)
	Telegram Event:  	
	
	\xFD 12345.BRS.23.STATUS.P1.P2 \xFE
	
		Funktionstyp:			BRS (kurz für Brightness Sensor)
		Instanz-ID:				hier 23 (in XML nachschauen)
		Aktion:					STATUS
		P1:						Relative Helligkeit 0-255 Vorkommastellen
		P2:						Relative Helligkeit 0-255 Nachkommastellen
	
	Telegram Statusabfrage:  	
	
	\xFD 12345.BRS.23.gSTATUS \xFE
	
	Antwort:  					\xFD 12345.BRS.23.rSTATUS.P1 \xFE
	P1:							Relative Helligkeit 0-255 Vorkommastellen
	P2:							Relative Helligkeit 0-255 Nachkommastellen

(*======================================================================================================================================*)
(* Alle Telegramme im Überblick *)	

	<?xml version="1.0" encoding="utf-8"?>
	<Comm Title="Haus-Bus ID 1212" Comment="" Baudrate="57600" Databits="8" Parity="1" EndChar="510">
	<CommCmd Title="16-fach Relais 1212 - Rote Modul LED" Comment="" CmdOn="\xFD1212.OUT.210.ON.0\xFE" CmdOff="\xFD1212.OUT.210.OFF\xFE" Unit="" Analog="false" Text="false" Sensor="false" SourceValHigh="100" DestValHigh="100"/>
	<CommCmd Title="16-fach Relais 1212 - Relais 1" Comment="" CmdOn="\xFD1212.OUT.17.ON.0\xFE" CmdOff="\xFD1212.OUT.17.OFF\xFE" Unit="" Analog="false" Text="false" Sensor="false" SourceValHigh="100" DestValHigh="100"/>
	<CommCmd Title="16-fach Relais 1212 - Relais 2" Comment="" CmdOn="\xFD1212.OUT.18.ON.0\xFE" CmdOff="\xFD1212.OUT.18.OFF\xFE" Unit="" Analog="false" Text="false" Sensor="false" SourceValHigh="100" DestValHigh="100"/>
	<CommCmd Title="16-fach Relais 1212 - Relais 3" Comment="" CmdOn="\xFD1212.OUT.19.ON.0\xFE" CmdOff="\xFD1212.OUT.19.OFF\xFE" Unit="" Analog="false" Text="false" Sensor="false" SourceValHigh="100" DestValHigh="100"/>
	<CommCmd Title="16-fach Relais 1212 - Relais 4" Comment="" CmdOn="\xFD1212.OUT.20.ON.0\xFE" CmdOff="\xFD1212.OUT.20.OFF\xFE" Unit="" Analog="false" Text="false" Sensor="false" SourceValHigh="100" DestValHigh="100"/>
	<CommCmd Title="16-fach Relais 1212 - Relais 5" Comment="" CmdOn="\xFD1212.OUT.21.ON.0\xFE" CmdOff="\xFD1212.OUT.21.OFF\xFE" Unit="" Analog="false" Text="false" Sensor="false" SourceValHigh="100" DestValHigh="100"/>
	<CommCmd Title="16-fach Relais 1212 - Relais 6" Comment="" CmdOn="\xFD1212.OUT.22.ON.0\xFE" CmdOff="\xFD1212.OUT.22.OFF\xFE" Unit="" Analog="false" Text="false" Sensor="false" SourceValHigh="100" DestValHigh="100"/>
	<CommCmd Title="16-fach Relais 1212 - Relais 7" Comment="" CmdOn="\xFD1212.OUT.23.ON.0\xFE" CmdOff="\xFD1212.OUT.23.OFF\xFE" Unit="" Analog="false" Text="false" Sensor="false" SourceValHigh="100" DestValHigh="100"/>
	<CommCmd Title="16-fach Relais 1212 - Relais 8" Comment="" CmdOn="\xFD1212.OUT.24.ON.0\xFE" CmdOff="\xFD1212.OUT.24.OFF\xFE" Unit="" Analog="false" Text="false" Sensor="false" SourceValHigh="100" DestValHigh="100"/>
	<CommCmd Title="16-fach Relais 1212 - Relais 9" Comment="" CmdOn="\xFD1212.OUT.33.ON.0\xFE" CmdOff="\xFD1212.OUT.33.OFF\xFE" Unit="" Analog="false" Text="false" Sensor="false" SourceValHigh="100" DestValHigh="100"/>
	<CommCmd Title="16-fach Relais 1212 - Relais 10" Comment="" CmdOn="\xFD1212.OUT.34.ON.0\xFE" CmdOff="\xFD1212.OUT.34.OFF\xFE" Unit="" Analog="false" Text="false" Sensor="false" SourceValHigh="100" DestValHigh="100"/>
	<CommCmd Title="16-fach Relais 1212 - Relais 11" Comment="" CmdOn="\xFD1212.OUT.35.ON.0\xFE" CmdOff="\xFD1212.OUT.35.OFF\xFE" Unit="" Analog="false" Text="false" Sensor="false" SourceValHigh="100" DestValHigh="100"/>
	<CommCmd Title="16-fach Relais 1212 - Relais 12" Comment="" CmdOn="\xFD1212.OUT.36.ON.0\xFE" CmdOff="\xFD1212.OUT.36.OFF\xFE" Unit="" Analog="false" Text="false" Sensor="false" SourceValHigh="100" DestValHigh="100"/>
	<CommCmd Title="16-fach Relais 1212 - Relais 13" Comment="" CmdOn="\xFD1212.OUT.37.ON.0\xFE" CmdOff="\xFD1212.OUT.37.OFF\xFE" Unit="" Analog="false" Text="false" Sensor="false" SourceValHigh="100" DestValHigh="100"/>
	<CommCmd Title="16-fach Relais 1212 - Relais 14" Comment="" CmdOn="\xFD1212.OUT.38.ON.0\xFE" CmdOff="\xFD1212.OUT.38.OFF\xFE" Unit="" Analog="false" Text="false" Sensor="false" SourceValHigh="100" DestValHigh="100"/>
	<CommCmd Title="16-fach Relais 1212 - Relais 15" Comment="" CmdOn="\xFD1212.OUT.39.ON.0\xFE" CmdOff="\xFD1212.OUT.39.OFF\xFE" Unit="" Analog="false" Text="false" Sensor="false" SourceValHigh="100" DestValHigh="100"/>
	<CommCmd Title="16-fach Relais 1212 - Relais 16" Comment="" CmdOn="\xFD1212.OUT.40.ON.0\xFE" CmdOff="\xFD1212.OUT.40.OFF\xFE" Unit="" Analog="false" Text="false" Sensor="false" SourceValHigh="100" DestValHigh="100"/>
	<CommCmd Title="16-fach Relais 1212 - Eingang 1" Comment="" CmdOn="\xFD1212.BTN.97.STATUS.\v\xFE" CmdOff="" Unit="&lt;v.x&gt;" Analog="true" Text="false" Sensor="true" SourceValHigh="100" DestValHigh="100"/>
	<CommCmd Title="16-fach Relais 1212 - Eingang 2" Comment="" CmdOn="\xFD1212.BTN.98.STATUS.\v\xFE" CmdOff="" Unit="&lt;v.x&gt;" Analog="true" Text="false" Sensor="true" SourceValHigh="100" DestValHigh="100"/>
	<CommCmd Title="16-fach Relais 1212 - Eingang 3" Comment="" CmdOn="\xFD1212.BTN.99.STATUS.\v\xFE" CmdOff="" Unit="&lt;v.x&gt;" Analog="true" Text="false" Sensor="true" SourceValHigh="100" DestValHigh="100"/>
	<CommCmd Title="16-fach Relais 1212 - Eingang 4" Comment="" CmdOn="\xFD1212.BTN.100.STATUS.\v\xFE" CmdOff="" Unit="&lt;v.x&gt;" Analog="true" Text="false" Sensor="true" SourceValHigh="100" DestValHigh="100"/>
	<CommCmd Title="16-fach Relais 1212 - Eingang 5" Comment="" CmdOn="\xFD1212.BTN.101.STATUS.\v\xFE" CmdOff="" Unit="&lt;v.x&gt;" Analog="true" Text="false" Sensor="true" SourceValHigh="100" DestValHigh="100"/>
	<CommCmd Title="16-fach Relais 1212 - Eingang 6" Comment="" CmdOn="\xFD1212.BTN.102.STATUS.\v\xFE" CmdOff="" Unit="&lt;v.x&gt;" Analog="true" Text="false" Sensor="true" SourceValHigh="100" DestValHigh="100"/>
	<CommCmd Title="16-fach Relais 1212 - Eingang 7" Comment="" CmdOn="\xFD1212.BTN.103.STATUS.\v\xFE" CmdOff="" Unit="&lt;v.x&gt;" Analog="true" Text="false" Sensor="true" SourceValHigh="100" DestValHigh="100"/>
	<CommCmd Title="16-fach Relais 1212 - Eingang 8" Comment="" CmdOn="\xFD1212.BTN.104.STATUS.\v\xFE" CmdOff="" Unit="&lt;v.x&gt;" Analog="true" Text="false" Sensor="true" SourceValHigh="100" DestValHigh="100"/>
	</Comm>

*)
END_ACTION

END_FUNCTION_BLOCK

// ---- POUs/RS485_Hausbus_FB/RelaisModul/fb_StringConvRB16F.TcPOU
(*======================================================================================================================================*)
(*fb_StringConvRB16F:	Zusammensetzen des Strings für 16Fach Bus Relaismodul		*)
(*
Date          	| Version    	| created under        	| Author          	| Remark *)
(*====================================================================================================================================================*)
(*08/05/2025   	| 1.00      		| TC3		  		| N.Kersting       | first release *)
(*====================================================================================================================================================*)
FUNCTION_BLOCK fb_StringConvRB16F
VAR_INPUT
	I_bReset			:BOOL;							(* Reset Befehl auslösen *)
	I_bRedLEDOn			:BOOL;							(* Schaltet nur die Rote Modul LED ein*)
	I_bRedLEDOff		:BOOL;							(* Schaltet nur die Rote Modul LED aus*)
	I_diID				:DINT;							(* Device ID *)
	I_bOut    	 		:ARRAY[1..16] OF BOOL;     	  	(* gewünschter Relais zustand (TRUE = An %)*)
	
	I_iSection			:INT :=1;							(* Paarweise Schalten 1= 1&2 2= 3&4 usw. *)
	
	I_sStartZeichen		:BYTE := 16#FD;					(* Startzeichen Präfix *)
	I_sEndZeichen		:BYTE := 16#FE;					(* Endzeichen Suffix *)
END_VAR
VAR_OUTPUT
	Q_sConvString		:STRING(255);
END_VAR
VAR
	iStartOut			:INT := 1;
	iStartInstIDExt		:INT :=65;
	
END_VAR

IF NOT I_bReset
THEN
	IF I_bRedLEDOn
	THEN
		(* Rote Modul LED Ein*)
		iStartInstIDExt := 210;
		
		Q_sConvString:=	CONCAT(F_ToCHR(I_sStartZeichen),DINT_TO_STRING(I_diID));
		Q_sConvString:=	CONCAT(Q_sConvString,'.OUT.');
		Q_sConvString:=	CONCAT(Q_sConvString,INT_TO_STRING(iStartInstIDExt));
		Q_sConvString:=	CONCAT(Q_sConvString,'.ON');
		Q_sConvString:=	CONCAT(Q_sConvString,F_ToCHR(I_sEndZeichen));
	ELSIF
		I_bRedLEDOff
	THEN
		(* Rote Modul LED Aus*)
		iStartInstIDExt := 210;
		
		Q_sConvString:=	CONCAT(F_ToCHR(I_sStartZeichen),DINT_TO_STRING(I_diID));
		Q_sConvString:=	CONCAT(Q_sConvString,'.OUT.');
		Q_sConvString:=	CONCAT(Q_sConvString,INT_TO_STRING(iStartInstIDExt));
		Q_sConvString:=	CONCAT(Q_sConvString,'.OFF');
		Q_sConvString:=	CONCAT(Q_sConvString,F_ToCHR(I_sEndZeichen));
	ELSE
		CASE I_iSection OF
			
		0:	Q_sConvString:='';
		
		1:	(* 1 & 2 Schalten *)
			iStartInstIDExt := 17;
			iStartOut :=	1;
			
			Q_sConvString:=	CONCAT(F_ToCHR(I_sStartZeichen),DINT_TO_STRING(I_diID));
			Q_sConvString:=	CONCAT(Q_sConvString,'.OUT.');
			Q_sConvString:=	CONCAT(Q_sConvString,INT_TO_STRING(iStartInstIDExt));
			IF I_bOut[iStartOut]
			THEN
				Q_sConvString:=	CONCAT(Q_sConvString,'.ON');
			ELSE
				Q_sConvString:=	CONCAT(Q_sConvString,'.OFF');
			END_IF
			Q_sConvString:=	CONCAT(Q_sConvString,F_ToCHR(I_sEndZeichen));
			
			(* ##2 ##*)
			iStartInstIDExt := iStartInstIDExt +1;
			iStartOut:= iStartOut+1;
			
			Q_sConvString:=	CONCAT(Q_sConvString,F_ToCHR(I_sStartZeichen));
			Q_sConvString:=	CONCAT(Q_sConvString,DINT_TO_STRING(I_diID));
			Q_sConvString:=	CONCAT(Q_sConvString,'.OUT.');
			Q_sConvString:=	CONCAT(Q_sConvString,INT_TO_STRING(iStartInstIDExt));
			IF I_bOut[iStartOut]
			THEN
				Q_sConvString:=	CONCAT(Q_sConvString,'.ON');
			ELSE
				Q_sConvString:=	CONCAT(Q_sConvString,'.OFF');
			END_IF
			Q_sConvString:=	CONCAT(Q_sConvString,F_ToCHR(I_sEndZeichen));
		
			(* ##3 ##*)
			iStartInstIDExt := iStartInstIDExt +1;
			iStartOut:= iStartOut+1;
			
			Q_sConvString:=	CONCAT(Q_sConvString,F_ToCHR(I_sStartZeichen));
			Q_sConvString:=	CONCAT(Q_sConvString,DINT_TO_STRING(I_diID));
			Q_sConvString:=	CONCAT(Q_sConvString,'.OUT.');
			Q_sConvString:=	CONCAT(Q_sConvString,INT_TO_STRING(iStartInstIDExt));
			IF I_bOut[iStartOut]
			THEN
				Q_sConvString:=	CONCAT(Q_sConvString,'.ON');
			ELSE
				Q_sConvString:=	CONCAT(Q_sConvString,'.OFF');
			END_IF
			Q_sConvString:=	CONCAT(Q_sConvString,F_ToCHR(I_sEndZeichen));
			
			(* ##4 ##*)
			iStartInstIDExt := iStartInstIDExt +1;
			iStartOut:= iStartOut+1;
			
			Q_sConvString:=	CONCAT(Q_sConvString,F_ToCHR(I_sStartZeichen));
			Q_sConvString:=	CONCAT(Q_sConvString,DINT_TO_STRING(I_diID));
			Q_sConvString:=	CONCAT(Q_sConvString,'.OUT.');
			Q_sConvString:=	CONCAT(Q_sConvString,INT_TO_STRING(iStartInstIDExt));
			IF I_bOut[iStartOut]
			THEN
				Q_sConvString:=	CONCAT(Q_sConvString,'.ON');
			ELSE
				Q_sConvString:=	CONCAT(Q_sConvString,'.OFF');
			END_IF
			Q_sConvString:=	CONCAT(Q_sConvString,F_ToCHR(I_sEndZeichen));
		
			(* ##5 ##*)
			iStartInstIDExt := iStartInstIDExt +1;
			iStartOut:= iStartOut+1;
			
			Q_sConvString:=	CONCAT(Q_sConvString,F_ToCHR(I_sStartZeichen));
			Q_sConvString:=	CONCAT(Q_sConvString,DINT_TO_STRING(I_diID));
			Q_sConvString:=	CONCAT(Q_sConvString,'.OUT.');
			Q_sConvString:=	CONCAT(Q_sConvString,INT_TO_STRING(iStartInstIDExt));
			IF I_bOut[iStartOut]
			THEN
				Q_sConvString:=	CONCAT(Q_sConvString,'.ON');
			ELSE
				Q_sConvString:=	CONCAT(Q_sConvString,'.OFF');
			END_IF
			Q_sConvString:=	CONCAT(Q_sConvString,F_ToCHR(I_sEndZeichen));
			
			(* ##6 ##*)
			iStartInstIDExt := iStartInstIDExt +1;
			iStartOut:= iStartOut+1;
			
			Q_sConvString:=	CONCAT(Q_sConvString,F_ToCHR(I_sStartZeichen));
			Q_sConvString:=	CONCAT(Q_sConvString,DINT_TO_STRING(I_diID));
			Q_sConvString:=	CONCAT(Q_sConvString,'.OUT.');
			Q_sConvString:=	CONCAT(Q_sConvString,INT_TO_STRING(iStartInstIDExt));
			IF I_bOut[iStartOut]
			THEN
				Q_sConvString:=	CONCAT(Q_sConvString,'.ON');
			ELSE
				Q_sConvString:=	CONCAT(Q_sConvString,'.OFF');
			END_IF
			Q_sConvString:=	CONCAT(Q_sConvString,F_ToCHR(I_sEndZeichen));
		
			(* ##7 ##*)
			iStartInstIDExt := iStartInstIDExt +1;
			iStartOut:= iStartOut+1;
			
			Q_sConvString:=	CONCAT(Q_sConvString,F_ToCHR(I_sStartZeichen));
			Q_sConvString:=	CONCAT(Q_sConvString,DINT_TO_STRING(I_diID));
			Q_sConvString:=	CONCAT(Q_sConvString,'.OUT.');
			Q_sConvString:=	CONCAT(Q_sConvString,INT_TO_STRING(iStartInstIDExt));
			IF I_bOut[iStartOut]
			THEN
				Q_sConvString:=	CONCAT(Q_sConvString,'.ON');
			ELSE
				Q_sConvString:=	CONCAT(Q_sConvString,'.OFF');
			END_IF
			Q_sConvString:=	CONCAT(Q_sConvString,F_ToCHR(I_sEndZeichen));
			
			(* ##8 ##*)
			iStartInstIDExt := iStartInstIDExt +1;
			iStartOut:= iStartOut+1;
			
			Q_sConvString:=	CONCAT(Q_sConvString,F_ToCHR(I_sStartZeichen));
			Q_sConvString:=	CONCAT(Q_sConvString,DINT_TO_STRING(I_diID));
			Q_sConvString:=	CONCAT(Q_sConvString,'.OUT.');
			Q_sConvString:=	CONCAT(Q_sConvString,INT_TO_STRING(iStartInstIDExt));
			IF I_bOut[iStartOut]
			THEN
				Q_sConvString:=	CONCAT(Q_sConvString,'.ON');
			ELSE
				Q_sConvString:=	CONCAT(Q_sConvString,'.OFF');
			END_IF
			Q_sConvString:=	CONCAT(Q_sConvString,F_ToCHR(I_sEndZeichen));
		
		2:	(* 9 & 10 Schalten *)
			iStartInstIDExt := 33;
			iStartOut :=	9;
			
			Q_sConvString:=	CONCAT(F_ToCHR(I_sStartZeichen),DINT_TO_STRING(I_diID));
			Q_sConvString:=	CONCAT(Q_sConvString,'.OUT.');
			Q_sConvString:=	CONCAT(Q_sConvString,INT_TO_STRING(iStartInstIDExt));
			IF I_bOut[iStartOut]
			THEN
				Q_sConvString:=	CONCAT(Q_sConvString,'.ON');
			ELSE
				Q_sConvString:=	CONCAT(Q_sConvString,'.OFF');
			END_IF
			Q_sConvString:=	CONCAT(Q_sConvString,F_ToCHR(I_sEndZeichen));
			
			(* ##10 ##*)
			iStartInstIDExt := iStartInstIDExt +1;
			iStartOut:= iStartOut+1;
			
			Q_sConvString:=	CONCAT(Q_sConvString,F_ToCHR(I_sStartZeichen));
			Q_sConvString:=	CONCAT(Q_sConvString,DINT_TO_STRING(I_diID));
			Q_sConvString:=	CONCAT(Q_sConvString,'.OUT.');
			Q_sConvString:=	CONCAT(Q_sConvString,INT_TO_STRING(iStartInstIDExt));
			IF I_bOut[iStartOut]
			THEN
				Q_sConvString:=	CONCAT(Q_sConvString,'.ON');
			ELSE
				Q_sConvString:=	CONCAT(Q_sConvString,'.OFF');
			END_IF
			Q_sConvString:=	CONCAT(Q_sConvString,F_ToCHR(I_sEndZeichen));
		
			(* ##11 ##*)
			iStartInstIDExt := iStartInstIDExt +1;
			iStartOut:= iStartOut+1;
			
			Q_sConvString:=	CONCAT(Q_sConvString,F_ToCHR(I_sStartZeichen));
			Q_sConvString:=	CONCAT(Q_sConvString,DINT_TO_STRING(I_diID));
			Q_sConvString:=	CONCAT(Q_sConvString,'.OUT.');
			Q_sConvString:=	CONCAT(Q_sConvString,INT_TO_STRING(iStartInstIDExt));
			IF I_bOut[iStartOut]
			THEN
				Q_sConvString:=	CONCAT(Q_sConvString,'.ON');
			ELSE
				Q_sConvString:=	CONCAT(Q_sConvString,'.OFF');
			END_IF
			Q_sConvString:=	CONCAT(Q_sConvString,F_ToCHR(I_sEndZeichen));
			
			(* ##12 ##*)
			iStartInstIDExt := iStartInstIDExt +1;
			iStartOut:= iStartOut+1;
			
			Q_sConvString:=	CONCAT(Q_sConvString,F_ToCHR(I_sStartZeichen));
			Q_sConvString:=	CONCAT(Q_sConvString,DINT_TO_STRING(I_diID));
			Q_sConvString:=	CONCAT(Q_sConvString,'.OUT.');
			Q_sConvString:=	CONCAT(Q_sConvString,INT_TO_STRING(iStartInstIDExt));
			IF I_bOut[iStartOut]
			THEN
				Q_sConvString:=	CONCAT(Q_sConvString,'.ON');
			ELSE
				Q_sConvString:=	CONCAT(Q_sConvString,'.OFF');
			END_IF
			Q_sConvString:=	CONCAT(Q_sConvString,F_ToCHR(I_sEndZeichen));
		
			(* ##13 ##*)
			iStartInstIDExt := iStartInstIDExt +1;
			iStartOut:= iStartOut+1;
			
			Q_sConvString:=	CONCAT(Q_sConvString,F_ToCHR(I_sStartZeichen));
			Q_sConvString:=	CONCAT(Q_sConvString,DINT_TO_STRING(I_diID));
			Q_sConvString:=	CONCAT(Q_sConvString,'.OUT.');
			Q_sConvString:=	CONCAT(Q_sConvString,INT_TO_STRING(iStartInstIDExt));
			IF I_bOut[iStartOut]
			THEN
				Q_sConvString:=	CONCAT(Q_sConvString,'.ON');
			ELSE
				Q_sConvString:=	CONCAT(Q_sConvString,'.OFF');
			END_IF
			Q_sConvString:=	CONCAT(Q_sConvString,F_ToCHR(I_sEndZeichen));
			
			(* ##14 ##*)
			iStartInstIDExt := iStartInstIDExt +1;
			iStartOut:= iStartOut+1;
			
			Q_sConvString:=	CONCAT(Q_sConvString,F_ToCHR(I_sStartZeichen));
			Q_sConvString:=	CONCAT(Q_sConvString,DINT_TO_STRING(I_diID));
			Q_sConvString:=	CONCAT(Q_sConvString,'.OUT.');
			Q_sConvString:=	CONCAT(Q_sConvString,INT_TO_STRING(iStartInstIDExt));
			IF I_bOut[iStartOut]
			THEN
				Q_sConvString:=	CONCAT(Q_sConvString,'.ON');
			ELSE
				Q_sConvString:=	CONCAT(Q_sConvString,'.OFF');
			END_IF
			Q_sConvString:=	CONCAT(Q_sConvString,F_ToCHR(I_sEndZeichen));
		
			(* ##15 ##*)
			iStartInstIDExt := iStartInstIDExt +1;
			iStartOut:= iStartOut+1;
			
			Q_sConvString:=	CONCAT(Q_sConvString,F_ToCHR(I_sStartZeichen));
			Q_sConvString:=	CONCAT(Q_sConvString,DINT_TO_STRING(I_diID));
			Q_sConvString:=	CONCAT(Q_sConvString,'.OUT.');
			Q_sConvString:=	CONCAT(Q_sConvString,INT_TO_STRING(iStartInstIDExt));
			IF I_bOut[iStartOut]
			THEN
				Q_sConvString:=	CONCAT(Q_sConvString,'.ON');
			ELSE
				Q_sConvString:=	CONCAT(Q_sConvString,'.OFF');
			END_IF
			Q_sConvString:=	CONCAT(Q_sConvString,F_ToCHR(I_sEndZeichen));
			
			(* ##16 ##*)
			iStartInstIDExt := iStartInstIDExt +1;
			iStartOut:= iStartOut+1;
			
			Q_sConvString:=	CONCAT(Q_sConvString,F_ToCHR(I_sStartZeichen));
			Q_sConvString:=	CONCAT(Q_sConvString,DINT_TO_STRING(I_diID));
			Q_sConvString:=	CONCAT(Q_sConvString,'.OUT.');
			Q_sConvString:=	CONCAT(Q_sConvString,INT_TO_STRING(iStartInstIDExt));
			IF I_bOut[iStartOut]
			THEN
				Q_sConvString:=	CONCAT(Q_sConvString,'.ON');
			ELSE
				Q_sConvString:=	CONCAT(Q_sConvString,'.OFF');
			END_IF
			Q_sConvString:=	CONCAT(Q_sConvString,F_ToCHR(I_sEndZeichen));
		END_CASE
	END_IF
	
ELSE
	(* Reset *)
	Q_sConvString:=	CONCAT(F_ToCHR(I_sStartZeichen),DINT_TO_STRING(I_diID));
	Q_sConvString:=	CONCAT(Q_sConvString,'.SYS.');
	Q_sConvString:=	CONCAT(Q_sConvString,INT_TO_STRING(1));
	Q_sConvString:=	CONCAT(Q_sConvString,'.RESET');
	Q_sConvString:=	CONCAT(Q_sConvString,F_ToCHR(I_sEndZeichen));
END_IF

END_FUNCTION_BLOCK

// ---- POUs/RS485_Hausbus_FB/CYD/fb_CYDBus6F.TcPOU
(*======================================================================================================================================*)
(*FB_TasterBusSimple:	Einfache RS485 Kommunikation für Haus-bus.de Komponenten zum testen 	
						Achtung: Bei dem 6 Fach Taster ist zu Beachten, dass es nur 4 Externe EA/s gibt also 4 LEDs und 4 Taster *)
(*
Date          	| Version    	| created under        	| Author          	| Remark *)
(*====================================================================================================================================================*)
(*29/04/2025   	| 1.00      		| TC3		  		| N.Kersting       | first release *)
(*02/05/2025   	| 1.01      		| TC3		  		| N.Kersting       | Events für die Buttons werden erfolgreich verarbeitet *)
(*02/05/2025   	| 1.02      		| TC3		  		| N.Kersting       | Events für Temp, Helligkeit, Fuehctigkeit erfolgreich Implementier *)
(*02/05/2025   	| 1.03      		| TC3		  		| N.Kersting       | Set Schrittkette für Reset und LED Helligkeit erfolgreich Implementier*)
(*02/05/2025   	| 1.04      		| TC3		  		| N.Kersting       | In und Out Strukturen Implementiert und Startup nach Reset *)
(*02/05/2025   	| 1.05      		| TC3		  		| N.Kersting       | Pingabgfrage*)
(*02/05/2025   	| 1.06      		| TC3		  		| N.Kersting       | Reset Startup Implementiert*)
(*03/05/2025   	| 1.07      		| TC3		  		| N.Kersting       | Ping wird nun bei PLC Reset auch gestaret und Execute wird richtig verwendet*)
(*04/05/2025   	| 1.08      		| TC3		  		| N.Kersting       | Hintergrundbeleuchtung und Zähler für die Tatser Implementiert *)
(*04/05/2025   	| 1.09      		| TC3		  		| N.Kersting       | Neuen Baustein zum Einheitlichen versenden von Telegrammen Implementiert *)
(*05/05/2025   	| 2.00      		| TC3		  		| N.Kersting       | Komplett neuen Baustein, mit Externer Receive Auswertung und neuem Ping Baustein *)
(*06/05/2025   	| 2.01      		| TC3		  		| N.Kersting       | Externe LEDs Implementiert *)
(*07/05/2025   	| 2.02      		| TC3		  		| N.Kersting       | Im Startup wird nun auf die Device ID geachtet *)
(*08/05/2025   	| 2.03      		| TC3		  		| N.Kersting       | Externe LEDs sind nun Umschaltbar/ LEDs oder normaler Ausgang (Betriefft die Hintergrundbeleuchtung) -> Weniger Busauslastung *)
(*09/05/2025   	| 2.04      		| TC3		  		| N.Kersting       | Ping Versuche Implementiert mit Globalen Parametern *)
(*09/05/2025   	| 2.05      		| TC3		  		| N.Kersting       | Ping für Taster nun Auch automatisch durch Empfang von sämtlichen Telegrammen*)
(*09/05/2025   	| 2.06      		| TC3		  		| N.Kersting       | Bugfix im Startup Angepasst! nur noch Hintergrundbeleuchtung setzen! *)
(*10/05/2025   	| 3.00      		| TC3		  		| N.Kersting       | Umstellung auf Externe FiFo Sendebaustein *)
(*13/05/2025   	| 3.01      		| TC3		  		| N.Kersting       | Viele Bugs gefixt, bei Änderung der Ausgängen wird nun eine Anforderung gesetzt  *)
(*13/05/2025   	| 3.02      		| TC3		  		| N.Kersting       | Test für Github *)
(*22/05/2025   	| 3.03      		| TC3		  		| N.Kersting       | Grundaufbau vom BusTaster, jetzt allerdings für ein CYD mit den gleichen Funktionen *)
(*22/05/2025   	| 3.04      		| TC3		  		| N.Kersting       | ServiceFunktionen für CYD Hinzugefügt (Wifi und Webserver Starten)*)
(*23/05/2025   	| 3.05      		| TC3		  		| N.Kersting       | Neue eigene Input Struktur für das CYD Implementiert*)
(*23/05/2025   	| 3.06      		| TC3		  		| N.Kersting       | Auto - Input Fault Detection implementiert (Wenn Taster zu lange aktiviert bleibt ) *)
(*26/05/2025   	| 3.07      		| TC3		  		| N.Kersting       | Updaten im Com Check Baustein, der Zyklische Ping vom CYD wird nun erkannt ) *)
(*28/05/2025   	| 3.08      		| TC3		  		| N.Kersting       | Neuen Einfachen Ping Baustein, welcher nicht sendet, nur auswertet implementiert *)
(*====================================================================================================================================================*)
FUNCTION_BLOCK fb_CYDBus6F
VAR_INPUT
	I_FifoID			:INT;
	I_bPingStart		:BOOL;						(* Ping Done vom Vorheriegen*)
	I_stInput			:ST_BusCYD6F_Input;
	I_StringReceived	:STRING(255);
END_VAR
VAR_OUTPUT
	Q_sFiFoSend			:STRING(255);
   	Q_stOutput			:ST_BusTaster6F_Output;
	Q_stCnt				:ST_BusTaster6F_Cnt;
END_VAR
VAR
(*----------------------------------------------*)
(* Interne Parameter*)
(*----------------------------------------------*)		
	bSetExecute			:BOOL := TRUE;				(* Aktiviert die Schrittketten, welche Telegramme versenden *)
	bCheckPing			:BOOL := TRUE;				(* Ping Checken Schrittkette Aktivieren *)
	sStartZeichen		:BYTE := 16#FD;				(* Startzeichen Präfix *)
	sEndZeichen			:BYTE := 16#FE;				(* Endzeichen Suffix *)
	iAnzResetSend		:INT := 2;					(* Anzahl der Sendeversuche bei Reset *)
	tPingTimer			:TIME:= T#5S;				(* Zeit, bis wiederholend der Ping versendet wird *)
	tReceiveTimeout		:TIME:= T#2S;				(* Zeit, bis die Event Schrittkette für das Empfangen Automatisch neu Startet*)
	tStartupLEDOn		:TIME:= T#4S;				(* Zeit, wie Lange die LEDS beim Startup kurz eingeschaltet werden *)
	tResetTimeout		:TIME:= T#25S;				(* Zeit, bis bei einem Reset es zu einem Fehler kommt, wenn kein Ping empfangen wird *)
	tResetReboot		:TIME:= T#10S;				(* Zeit, die nach einem Reset Abgewaretet wird damit das Gerät neustarten kann*)
	tResetStartup		:TIME:= T#5S;				(* Zeit, die nach einem Reset Abgewaretet wird bis ein Startup ausgeführt wird nach dem erhalt des Pings vom Gerät*)
	tStartupAfterReset	:TIME := T#5S;				(* Zeit, wann das Startup Zurückgesetzt wird, wenn der Ping verloren wird *)
	bInputFaultDetect	:BOOL := TRUE;				(* Prüft die Eingänge ob sie zu lange geschaltet wurden und führt ein reset des eingangs aus *)
	tInputFaultDetect	:TIME := T#10S;				(* Prüft die Eingänge ob sie zu lange geschaltet wurden und führt ein reset des eingangs aus *)
(*----------------------------------------------*)
(*	Service Funktionen Aktivieren *)
(*----------------------------------------------*)	
	bWebServer			:BOOL := FALSE;				(* zuerst funktion auswählen (bWebserver/ bWifi, bService) und dann mit bStartServiceMode ausführen *)
	bWifi				:BOOL := FALSE;				(* zuerst funktion auswählen (bWebserver/ bWifi, bService) und dann mit bStartServiceMode ausführen *)
	bService			:BOOL := FALSE;				(* zuerst funktion auswählen (bWebserver/ bWifi, bService) und dann mit bStartServiceMode ausführen *)
	(*	*)
	bStartServiceMode	:BOOL := FALSE;				(* zuerst ServiceMode Aktivieren und dann mit bStartServiceMode ausführen *)
	
	(* Speichern der zustände *)
	bMemWebServer		:BOOL;
	bMemWifi			:BOOL;
	bMemService			:BOOL;
	
(*----------------------------------------------*)
(* Strings *)
(*----------------------------------------------*)			
	sSendString			:STRING(255);
	sFiFoSend			:STRING(255);
	sReceived			:STRING(255);
	sLastSendString		:STRING(255);
	sStateReset			:STRING;
(*----------------------------------------------*)
(* Funktionsbausteine *)
(*----------------------------------------------*)
	fbBusTasterEvent	:ARRAY[1..6] OF fb_BusTasterEvent;		(* Interne 6 Taster Abfragen *)
	fbBusTasterEventExt	:ARRAY[1..6] OF fb_BusTasterEvent;		(* Externe 6 Eingänge Abfragen *)
	fbBusTempEvent		:fb_BusTempEvent;
	fbBusBrsEvent		:fb_BusBrsEvent;
	fbBusRhdEvent		:fb_BusRhdEvent;
	fbStringConvTB6F	:fb_StringConvTB6F;
	fbStringConvWeb		:fb_StringConvCYDWeb;
	fbStringConvWifi	:fb_StringConvCYDWifi;
	fbStringConvService	:fb_StringConvCYDService;
	fbPing				:fb_RS485Ping;
(*----------------------------------------------*)
(* Indexe *)
(*----------------------------------------------*)	
	iDeviceStartup		:INT :=0;	(* Startup Schrittkette *)
	sDeviceStartup		:STRING;
    iState     			:INT := 0;
	iStepSet			:INT;
	i,h,j,l,e			:INT;
	idxLED				:INT;
	idxBtn				:INT := 1;
	
	iDimmMem			:ARRAY[1..6] OF INT;
	iDimmMemExt			:ARRAY[1..6] OF INT;
	iDimmBGAnf			:INT;
	iDimmAnf			:ARRAY[1..6] OF INT;
	iDimmAnfExt			:ARRAY[1..6] OF INT;
	
	iDimmBgMem			:INT;
	cntChangesDimm		:INT;
	cntChangesDimmExt	:INT;
	icntResetSend		:INT;
	iMaxPingTry			:INT := 5;
(*----------------------------------------------*)
(* Timer/Trigger *)
(*----------------------------------------------*)		
	r_trigStartupAfterReset	:r_trig;
	r_TrigReset				:r_trig;		
	r_TrigCountBtn			:ARRAY[1..6] OF r_trig;
	
	tonStartupAfterReset	:ton;
	tonReceiveTimeout		:ton;
	tonResetTimeout			:ton;
	tonResetDone			:ton;
	tonStepStartup			:ton;
(*----------------------------------------------*)
(* Status *)
(*----------------------------------------------*)			
	bPingOK					:BOOL;
	bErrorEvent				:BOOL;
	bErrorPing				:BOOL;
	bErrorSet				:BOOL;
	bErrorReset				:BOOL;
	bResetBusy				:BOOL;
	bResetDone				:BOOL;
	bResetAutoStart			:BOOL;
	bStartupStart			:BOOL;
	bStartupDone			:BOOL;	
	bMemExt					:BOOL;
	bStartUpCheckPing		:BOOL;
	bActivateSend			:BOOL;
	bReadyToPing			:BOOL;
	bSendeAnforderung		:BOOL;
	bSendeAnforderungExt	:BOOL;
	bSendeAnforderungBG		:BOOL;
	
END_VAR

(*============================================================================================*)
(* Parameter *)
tPingTimer :=		GVL_HausBus_Parameter.cTimePingTimeCYD;
tReceiveTimeout :=	GVL_HausBus_Parameter.cTimeReceiveTimeoutCYD;
bCheckPing :=		GVL_HausBus_Parameter.bUseCYDPing;
iMaxPingTry :=		GVL_HausBus_Parameter.cMaxPingTry;

(* Service *)
bWebServer :=			I_stInput.bWebServer;
bWifi :=				I_stInput.bWifi;
bService :=				I_stInput.bService;
bStartServiceMode :=	I_stInput.bServiceMode;

(*============================================================================================*)
(* Startup Zurücksetzen Reset *)
r_TrigReset(CLK := I_stInput.bReset);

(* Startup Zurücksetzen bei Busverlust *)
tonStartupAfterReset(
	IN := NOT bPingOK
			AND bCheckPing,
	PT:= tStartupAfterReset);

r_trigStartupAfterReset
	(CLK := tonStartupAfterReset.Q);
	
IF NOT I_stInput.bExecute
	OR r_TrigReset.Q
	OR r_trigStartupAfterReset.Q
THEN
	iDeviceStartup := 0;
ELSIF
	bStartServiceMode
THEN	
	iDeviceStartup := 5;
END_IF

(*============================================================================================*)
(* Ping Dauerhaft Senden*)
ac02_Ping();
	
(*============================================================================================*)
(* Startup Schrittkette *)
CASE iDeviceStartup OF
(*============================================================================================*)
0: 	sDeviceStartup := 'INIT';
	bResetDone := FALSE;
	bStartupDone := FALSE;
	bStartupStart := FALSE;
	bResetAutoStart := FALSE;
	bStartUpCheckPing := FALSE;
	bActivateSend := FALSE;
	bReadyToPing := TRUE;
	bMemWebServer :=FALSE;
	bMemWifi :=	FALSE;
	bMemService	:= FALSE;
	
	sFiFoSend := ''; 
	iStepSet := 0;
	
	IF 	I_stInput.bExecute
	THEN
		iDeviceStartup := iDeviceStartup+1;
	END_IF
(*============================================================================================*)
1: 	sDeviceStartup := 'Device ID Prüfen';
	
	IF  I_stInput.diID <> 0
	THEN
		iDeviceStartup := iDeviceStartup+1;
	ELSE
		sDeviceStartup := 'ERROR- Device ID Prüfen';
	END_IF
(*============================================================================================*)
2: 	sDeviceStartup := 'Verbindung Prüfen';
	bActivateSend := TRUE;	(* Senden Aktivieren *)
	iDeviceStartup := iDeviceStartup+1;
	
	(*
	sDeviceStartup := CONCAT(sDeviceStartup,fbRS485ComCheck.Q_sState);
	
	IF fbRS485ComCheck.Q_bComOk
		OR NOT bCheckPing
	THEN
	END_IF*)

(*============================================================================================*)
3: 	sDeviceStartup := 'Reset Ausführen';	
	bActivateSend := TRUE;	(* Senden Aktivieren *)
	
	(*	RESET Device *)
	ac01_SetReset();
	bResetAutoStart := TRUE;
	
	sDeviceStartup :=	CONCAT(sDeviceStartup,sStateReset);
	
	IF bResetDone
	THEN
		iStepSet := 0;
		iDeviceStartup := iDeviceStartup+1;
	END_IF

(*============================================================================================*)
4: 	sDeviceStartup := 'Startup Ausführen';
		
	(* LED Setzen *)
	ac01_SetLED();
	
	bStartupStart := TRUE;
	
	IF bStartupDone 
	THEN
		bStartupStart := FALSE;
		iDeviceStartup := 999;
	END_IF

(*============================================================================================*)
5:	sDeviceStartup := 'Service Funktionen Steuern';
	ac01_SetService();

	IF NOT bStartServiceMode 
	THEN
		iStepSet := 0;
		iDeviceStartup := 0;
	END_IF
	
(*============================================================================================*)
999: 
	(*bReadyToPing := NOT fbRS485SendCmd.Q_bBusy;*)
	
	(* LED Setzen *)
	ac01_SetLED();
	
	(* Events Auslesen *)
	ac00_Event();
	
	(* Zähler *)
	ac10_Counter();
	
	sDeviceStartup := 'Startup Ausgeführt- Gerät im OP';
	
END_CASE

(*============================================================================================*)
(* Sendebaustein *)
IF bActivateSend
THEN
	Q_sFiFoSend :=	sFiFoSend;
END_IF

(*============================================================================================*)	
(* Zähler *)
ac10_Counter();
	
(*============================================================================================*)
(* Outputs *)
Q_stOutput.bCOM :=		bPingOK;

Q_stOutput.bError := 	bErrorEvent
						OR bErrorPing
						OR bErrorSet
						OR (NOT bPingOK
						AND bCheckPing);
						
Q_stOutput.bStartupDone	:=	bStartupDone;

Q_stOutput.sState :=	CONCAT(I_stInput.sName,'| ');
Q_stOutput.sState :=	CONCAT(Q_stOutput.sState, sDeviceStartup);

ACTION ac00_Event:
(*============================================================================================*)
(*	EVENT Schrittkette *)
(*============================================================================================*)
sReceived := I_StringReceived;
	
FOR i := 1 TO 6 BY 1 DO 
	fbBusTasterEvent[i](
		I_bFaultDetection	:=	bInputFaultDetect,
		I_tFaultDetectTime	:=	tInputFaultDetect,
		I_sID:= 				DINT_TO_STRING(I_stInput.diID), 
		I_sInstID:= 			INT_TO_STRING(i+16), 
		I_sReceivedString:= 	sReceived, 
		Q_bOut=> 				Q_stOutput.bButtons[i]);
	
	fbBusTasterEventExt[i](
		I_sID:= 				DINT_TO_STRING(I_stInput.diID), 
		I_sInstID:= 			INT_TO_STRING(i+32), 
		I_sReceivedString:= 	sReceived, 
		Q_bOut=> 				Q_stOutput.bButtonsExt[i]);
		
	fbBusTempEvent(
		I_sID:= 				DINT_TO_STRING(I_stInput.diID), 
		I_sInstID:= 			'1', 
		I_sReceivedString:= 	sReceived, 
		Q_lrTemp=> 				Q_stOutput.lrTemp);
		
	fbBusBrsEvent(
		I_sID:= 				DINT_TO_STRING(I_stInput.diID), 
		I_sInstID:= 			'1', 
		I_sReceivedString:= 	sReceived, 
		Q_lrBrs=> 				Q_stOutput.lrBrs);
		
	fbBusRhdEvent(
		I_sID:= 				DINT_TO_STRING(I_stInput.diID), 
		I_sInstID:= 			'1', 
		I_sReceivedString:= 	sReceived, 
		Q_lrRhd=> 				Q_stOutput.lrRhd);
END_FOR
END_ACTION

ACTION ac01_SetLED:
(*============================================================================================*)
(*	LED Helligkeit Setzen/ Startup Schrittkette *)
(*============================================================================================*)

(* Einfaches Setzen der LED Helligkeiten (0-100 Prozent *)
(* Neu, es werden alle LEDs zu einem String zusammengefügt und Gleichzeitig gesetzt *)
tonStepStartup(
	PT:= tStartupLEDOn);
	
cntchangesDimm := 0;
cntChangesDimmExt :=0;
	
FOR l := 1 TO 6 BY 1 DO
	IF iDimmMem[l] <> I_stInput.iLED[l]
	THEN
		cntChangesDimm := cntChangesDimm +1;
	END_IF

	IF  iDimmMemExt[l]<> I_stInput.iLEDExt[l]
	THEN
		cntChangesDimmExt := cntChangesDimmExt +1;
	END_IF
END_FOR

CASE iStepSet OF
(*============================================================================================*)
0:	(* INIT und warten auf Change *)				
	tonStepStartup.IN := FALSE;
	sFiFoSend := ''; 
	
	(* Änderungs- Anforderungen Prüfen*)
	FOR e := 1 TO 6 BY 1 DO
		IF cntChangesDimm<>0
		THEN
			(* Helligkeitanforderung Interne LEDs speichern *)
			bSendeAnforderung := TRUE;
			iDimmAnf[e] 	:= I_stInput.iLED[e];
		END_IF
		
		IF cntChangesDimmExt <> 0
		THEN
			(* Helligkeitanforderung Externe LEDs speichern *)
			bSendeAnforderungExt := TRUE;
			iDimmAnfExt[e] 	:= I_stInput.iLEDExt[e];
		END_IF
		
		IF I_stInput.iLEDBg <>iDimmBgMem
		THEN
			(* Helligkeitsanforderung Hintergrundbeleuchtung *)
			bSendeAnforderungBG := TRUE;
			iDimmBGAnf		:= I_stInput.iLEDBg;
		END_IF
	END_FOR
	
	(* Reagieren auf Anforderungen *)
	IF ((bSendeAnforderung
		OR bSendeAnforderungExt
		OR bSendeAnforderungBG)
		AND bSetExecute)
		AND NOT bStartupStart
	THEN
		(* Helligkeitsvorgaben speichern in Mem Arrays *)
		FOR h := 1 TO 6 BY 1 DO
			iDimmMem[h] := I_stInput.iLED[h];
			iDimmMemExt[h] := I_stInput.iLEDExt[h];
			iDimmBgMem := I_stInput.iLEDBg;
		END_FOR
		
		iStepSet := 10;
	ELSIF
		bStartupStart
	THEN
		iStepSet := 100;	(* Startup *)
	END_IF
	
(*============================================================================================*)
10:	(* Prüfen welche Anforderung ausgeführt werden soll *)	
	IF	bSendeAnforderungBG
		AND NOT bSendeAnforderung
		AND NOT bSendeAnforderungExt 
	THEN
		iStepSet := 22;(* Direkt nur die Hintergrund Helligkeit setzen *)
	ELSE
		(* Nur Interne LEDs Schreiben *)
		IF bSendeAnforderung
			AND NOT bSendeAnforderungExt
			AND NOT bSendeAnforderungBG
		THEN
			fbStringConvTB6F(
				I_bSetBackground :=	FALSE,
				I_bReset :=			FALSE,
				I_bExtLED :=		FALSE,
				I_bHasExtLED :=		I_stInput.bExtOutLED,
				I_diID:= 			I_stInput.diID, 
				I_iLED:= 			iDimmAnf, 
				I_iLEDExt:=			iDimmAnfExt,
				I_iLEDBg:= 			iDimmBGAnf,		 
				I_sStartZeichen:= 	sStartZeichen, 
				I_sEndZeichen:= 	sEndZeichen, 
				Q_sConvString=> 	sSendString);
				
			(* Senden an FiFo*)
			IF GVL_RS485FiFoSend.bSendDoneFiFo[I_FifoID]
			THEN
				sFiFoSend :=	sSendString;
			END_IF
			IF NOT GVL_RS485FiFoSend.bSendDoneFiFo[I_FifoID]
			THEN
				bSendeAnforderung := FALSE;
				sLastSendString :=	sFiFoSend;
				iStepSet := 20;
			END_IF
		ELSIF
			(* Nur Externe LEDs Schreiben *)	
			bSendeAnforderungExt
			AND NOT bSendeAnforderung
			AND NOT bSendeAnforderungBG
		THEN
			fbStringConvTB6F(
				I_bSetBackground :=	FALSE,
				I_bReset :=			FALSE,
				I_bExtLED :=		TRUE,
				I_bHasExtLED :=		I_stInput.bExtOutLED,
				I_diID:= 			I_stInput.diID, 
				I_iLED:= 			iDimmAnf, 
				I_iLEDExt:=			iDimmAnfExt,
				I_iLEDBg:= 			iDimmBGAnf,				 
				I_sStartZeichen:= 	sStartZeichen, 
				I_sEndZeichen:= 	sEndZeichen, 
				Q_sConvString=> 	sSendString);
			
			(* Senden an FiFo*)
			IF GVL_RS485FiFoSend.bSendDoneFiFo[I_FifoID]
			THEN
				sFiFoSend :=	sSendString;
			END_IF
			IF NOT GVL_RS485FiFoSend.bSendDoneFiFo[I_FifoID]
			THEN
				bSendeAnforderungExt := FALSE;
				sLastSendString :=	sFiFoSend;
				iStepSet := 20;
			END_IF
		ELSE
			(* Externe und Interne LEDs Schreiben *)
			bMemExt := TRUE; (* Speichern, damit anschließend noch die Externen LEDs gesetzt werden *)
			
			fbStringConvTB6F(
				I_bSetBackground :=	FALSE,
				I_bReset :=			FALSE,
				I_bExtLED :=		FALSE,
				I_bHasExtLED :=		I_stInput.bExtOutLED,
				I_diID:= 			I_stInput.diID, 
				I_iLED:= 			iDimmAnf, 
				I_iLEDExt:=			iDimmAnfExt,
				I_iLEDBg:= 			iDimmBGAnf,			 
				I_sStartZeichen:= 	sStartZeichen, 
				I_sEndZeichen:= 	sEndZeichen, 
				Q_sConvString=> 	sSendString);
			
			(* Senden an FiFo*)
			IF GVL_RS485FiFoSend.bSendDoneFiFo[I_FifoID]
			THEN
				sFiFoSend :=	sSendString;
			END_IF
			IF NOT GVL_RS485FiFoSend.bSendDoneFiFo[I_FifoID]
			THEN
				bSendeAnforderung := FALSE;
				bSendeAnforderungExt := FALSE;
				sLastSendString :=	sFiFoSend;
				iStepSet := 20;
			END_IF
		END_IF
	END_IF
(*============================================================================================*)	
20:	(* Warten bis nicht Busy *)	
	
	IF GVL_RS485FiFoSend.bSendDoneFiFo[I_FifoID]
	THEN
		sFiFoSend := ''; 
		IF NOT bMemExt
		THEN
			IF bSendeAnforderungBG
			THEN
				iStepSet := 22;
			ELSE
				iStepSet := 0;
			END_IF
		ELSE
			iStepSet :=	21;
		END_IF
	END_IF
	
(*============================================================================================*)	
21:	(* Externe LEDs Senden *)	
	bMemExt := FALSE;
	bSendeAnforderungExt := FALSE;
	
	fbStringConvTB6F(
		I_bSetBackground :=	FALSE,
		I_bReset :=			FALSE,
		I_bExtLED :=		TRUE,
		I_bHasExtLED :=		I_stInput.bExtOutLED,
		I_diID:= 			I_stInput.diID, 
		I_iLED:= 			iDimmAnf, 
		I_iLEDExt:=			iDimmAnfExt,
		I_iLEDBg:= 			iDimmBGAnf,				 
		I_sStartZeichen:= 	sStartZeichen, 
		I_sEndZeichen:= 	sEndZeichen, 
		Q_sConvString=> 	sSendString);
		
	(* Senden an FiFo*)
	IF GVL_RS485FiFoSend.bSendDoneFiFo[I_FifoID]
	THEN
		sFiFoSend :=	sSendString;
	END_IF
	IF NOT GVL_RS485FiFoSend.bSendDoneFiFo[I_FifoID]
	THEN
		sLastSendString :=	sFiFoSend;
		iStepSet := 20;
	END_IF
	
(*============================================================================================*)	
22:	(* Hintergrundbeleuchtung senden *)		
	bSendeAnforderungBG := FALSE;
	
	fbStringConvTB6F(
		I_bSetBackground :=	TRUE,
		I_bReset :=			FALSE,
		I_bExtLED :=		FALSE,
		I_bHasExtLED :=		I_stInput.bExtOutLED,
		I_diID:= 			I_stInput.diID, 
		I_iLED:= 			iDimmAnf, 
		I_iLEDExt:=			iDimmAnfExt,
		I_iLEDBg:= 			iDimmBGAnf,			 
		I_sStartZeichen:= 	sStartZeichen, 
		I_sEndZeichen:= 	sEndZeichen, 
		Q_sConvString=> 	sSendString);
		
	(* Senden an FiFo*)
	IF GVL_RS485FiFoSend.bSendDoneFiFo[I_FifoID]
	THEN
		sFiFoSend :=	sSendString;
	END_IF
	IF NOT GVL_RS485FiFoSend.bSendDoneFiFo[I_FifoID]
	THEN
		sLastSendString :=	sFiFoSend;
		iStepSet := 20;
	END_IF

(*============================================================================================*)	
(* Startup LEDS einmal Einschalten *)
100:	tonStepStartup.IN := TRUE;
	
	IF tonStepStartup.Q
	THEN
		iStepSet := 110;
	END_IF
	
(*============================================================================================*)
110:	(* String senden *)	
	tonStepStartup.IN := FALSE;
	
	fbStringConvTB6F(
		I_bSetBackground :=	TRUE,
		I_bExtLED :=		FALSE,
		I_bReset :=			FALSE,
		I_bHasExtLED :=		I_stInput.bExtOutLED,
		I_diID:= 			I_stInput.diID, 
		I_iLEDBg:= 			5,		 
		I_sStartZeichen:= 	sStartZeichen, 
		I_sEndZeichen:= 	sEndZeichen, 
		Q_sConvString=> 	sSendString);
			
	(* Senden an FiFo*)
	IF GVL_RS485FiFoSend.bSendDoneFiFo[I_FifoID]
	THEN
		sFiFoSend :=	sSendString;
	END_IF
	IF NOT GVL_RS485FiFoSend.bSendDoneFiFo[I_FifoID]
	THEN
		
		iStepSet := 111;
	END_IF
	
(*============================================================================================*)	
111:(* Warten bis nicht Busy *)	
	IF GVL_RS485FiFoSend.bSendDoneFiFo[I_FifoID]
	THEN
		sFiFoSend := ''; 
		tonStepStartup.IN := TRUE;
		
		IF tonStepStartup.Q
		THEN
			tonStepStartup.IN := FALSE;
			iStepSet := 120;
		END_IF
	END_IF
	
(*============================================================================================*)
120:	(* String senden *)	
	fbStringConvTB6F(
		I_bSetBackground :=	TRUE,
		I_bExtLED :=		FALSE,
		I_bReset :=			FALSE,
		I_bHasExtLED :=		I_stInput.bExtOutLED,
		I_diID:= 			I_stInput.diID, 
		I_iLEDBg:= 			100,		 
		I_sStartZeichen:= 	sStartZeichen, 
		I_sEndZeichen:= 	sEndZeichen, 
		Q_sConvString=> 	sSendString);
			
	(* Senden an FiFo*)
	IF GVL_RS485FiFoSend.bSendDoneFiFo[I_FifoID]
	THEN
		sFiFoSend :=	sSendString;
	END_IF
	IF NOT GVL_RS485FiFoSend.bSendDoneFiFo[I_FifoID]
	THEN
		iStepSet := 130;
	END_IF
	
(*============================================================================================*)	
130:(* Warten bis nicht Busy *)	
	IF GVL_RS485FiFoSend.bSendDoneFiFo[I_FifoID]
	THEN
		sFiFoSend := ''; 
			
		tonStepStartup.IN := TRUE;
	
		IF tonStepStartup.Q
		THEN
			bStartupDone := TRUE;
			tonStepStartup.IN := FALSE;
			bStartupStart := FALSE;
			iStepSet := 10;	(* Anschließend noch einmal die Eingangs Helligkeit setzen *)
		END_IF
	END_IF	

END_CASE

(*bErrorSet := fbRS485SendCmd.Q_bError;*)
END_ACTION

ACTION ac01_SetReset:
(*============================================================================================*)
(*	RESET Schrittkette *)
(*============================================================================================*)
tonResetTimeout(
	PT := tResetTimeout);

tonResetDone();

(* Einfaches Setzen der LED Helligkeiten (0-100 Prozent *)
CASE iStepSet OF
(*============================================================================================*)
0:	sStateReset := 'INIT';
	
	IF (bSetExecute
		AND (I_stInput.bReset
		OR bResetAutoStart))
	THEN
		sFiFoSend := ''; 
		bStartupDone := FALSE;
		bResetDone := FALSE;
		tonResetTimeout.IN := FALSE;
		tonResetDone.IN := FALSE;
		icntResetSend := 0;
		
		(* Ausgänge alle auf 0 setzen *)
		FOR h := 1 TO 6 BY 1 DO
			fbBusTasterEvent[i](
				I_sReceivedString :='');
				
			fbBusTasterEventExt[i](
				I_sReceivedString :='');	
				
			iDimmMem[h] := 0;
			Q_stOutput.bButtons[h] := FALSE;
			Q_stOutput.lrTemp := 0;
			Q_stOutput.lrBrs := 0;
			Q_stOutput.lrRhd := 0;
		END_FOR
		
		fbBusTempEvent(
			I_sReceivedString :='',	
			I_bReset := TRUE);
			
		fbBusBrsEvent(
			I_sReceivedString :='',	
			I_bReset := TRUE);
			
		fbBusRhdEvent(
			I_sReceivedString :='',	
			I_bReset := TRUE);
		
		bPingOK := FALSE;
		
		iStepSet := iStepSet +1;
	END_IF

(*============================================================================================*)	
1:	sStateReset := 'Sende Reset Befehl';
	bResetBusy := TRUE;
	bErrorReset := FALSE;
	
	fbStringConvTB6F(
		I_bReset :=			TRUE,
		I_diID:= 			I_stInput.diID, 		 
		I_sStartZeichen:= 	sStartZeichen, 
		I_sEndZeichen:= 	sEndZeichen, 
		Q_sConvString=> 	sSendString);

	(* Senden an FiFo*)
	IF GVL_RS485FiFoSend.bSendDoneFiFo[I_FifoID]
	THEN
		sFiFoSend :=	sSendString;
	END_IF
	IF NOT GVL_RS485FiFoSend.bSendDoneFiFo[I_FifoID]
	THEN
		iStepSet := iStepSet+1;
	END_IF

(*============================================================================================*)
2:	sStateReset := 'Sende Reset Befehl';

	IF GVL_RS485FiFoSend.bSendDoneFiFo[I_FifoID]
	THEN
		sFiFoSend := ''; 
		fbStringConvTB6F(
			I_bReset :=			FALSE);
		iStepSet := 3;
				
	END_IF
	
(*============================================================================================*)	
3:	sStateReset := 'Reset durchgeführt, Warte auf Ping';
	tonResetDone.IN := TRUE;
	tonResetDone.PT := tResetReboot;
	
	fbBusTempEvent(I_bReset := FALSE);
	fbBusBrsEvent(I_bReset := FALSE);
	fbBusRhdEvent(I_bReset := FALSE);
	
	iState := 0;
	
	IF tonResetDone.Q
	THEN
		tonResetDone.IN := FALSE;
		iStepSet := 4;
	END_IF
	
(*============================================================================================*)	
4:	sStateReset := 'Warte auf Ping vom Gerät';	
	tonResetTimeout.IN := TRUE;
	bStartUpCheckPing := TRUE;
	
	IF bPingOK 
	(*	OR NOT bCheckPing*)
	THEN
		bErrorReset := FALSE;
		tonResetTimeout.IN := FALSE;
		iStepSet := 5;
	ELSIF
		tonResetTimeout.Q
	THEN
		sStateReset := 'Ping Timeout, keine Kommunikation';
		bErrorReset := TRUE;

		IF I_stInput.bReset
		THEN
			bResetBusy := FALSE;
			iStepSet := 0;
		END_IF
	END_IF

(*============================================================================================*)
5:	sStateReset := 'Startup Aktiv';
	
	tonResetDone.IN := NOT I_stInput.bReset;
	tonResetDone.PT := tResetStartup;
	sFiFoSend := ''; 
	
	IF tonResetDone.Q
	THEN
		fbStringConvTB6F(
			I_bReset :=			FALSE);
			
		sStateReset := 'Ping erhalten, Reset Erfolgreich';
		bResetAutoStart := FALSE;
		bResetDone := TRUE;
		bResetBusy := FALSE;
		iState := 0;
		iStepSet := 0;
	END_IF
END_CASE
END_ACTION

ACTION ac01_SetService:
(*============================================================================================*)
(*	RESET Schrittkette *)
(*============================================================================================*)
tonResetTimeout(
	PT := tResetTimeout);

tonResetDone();

(* Einfaches Setzen der LED Helligkeiten (0-100 Prozent *)
CASE iStepSet OF
(*============================================================================================*)
0:	sStateReset := 'INIT';
	
	IF bSetExecute
		AND (bMemWebServer <> bWebServer
		OR bMemWifi <> bWifi
		OR bMemService <> bService )
	THEN
		bMemWebServer :=	bWebServer;
		bMemWifi :=			bWifi;
		bMemService	:=		bService;
		
		sFiFoSend := ''; 
		tonResetTimeout.IN := FALSE;
		tonResetDone.IN := FALSE;
		icntResetSend := 0;
		
		iStepSet := iStepSet +1;
	END_IF

(*============================================================================================*)	
1:	sStateReset := 'Sende Webserver Befehl';
	fbStringConvWeb(
		I_diID:= 			I_stInput.diID,
		I_bWebOn:= 			bWebServer, 
		I_sStartZeichen:= 	sStartZeichen, 
		I_sEndZeichen:= 	sEndZeichen, 
		Q_sConvString=> 	sSendString);
	
	(* Senden an FiFo*)
	IF GVL_RS485FiFoSend.bSendDoneFiFo[I_FifoID]
	THEN
		sFiFoSend :=	sSendString;
	END_IF
	IF NOT GVL_RS485FiFoSend.bSendDoneFiFo[I_FifoID]
	THEN
		iStepSet := iStepSet+1;
	END_IF

(*============================================================================================*)
2:	sStateReset := 'Sende Webserver Befehl';

	IF GVL_RS485FiFoSend.bSendDoneFiFo[I_FifoID]
	THEN
		sFiFoSend := ''; 
		iStepSet := 3;
	END_IF
	
(*============================================================================================*)	
3:	sStateReset := 'Sende Wifi Befehl';
	
	fbStringConvWifi(
		I_diID:= 			I_stInput.diID,
		I_bWifiOn:= 		bWifi, 
		I_sStartZeichen:= 	sStartZeichen, 
		I_sEndZeichen:= 	sEndZeichen, 
		Q_sConvString=> 	sSendString);
	
	(* Senden an FiFo*)
	IF GVL_RS485FiFoSend.bSendDoneFiFo[I_FifoID]
	THEN
		sFiFoSend :=	sSendString;
	END_IF
	IF NOT GVL_RS485FiFoSend.bSendDoneFiFo[I_FifoID]
	THEN
		iStepSet := iStepSet+1;
	END_IF
	
(*============================================================================================*)	
4:	sStateReset := 'Sende Wifi Befehl';

	IF GVL_RS485FiFoSend.bSendDoneFiFo[I_FifoID]
	THEN
		sFiFoSend := ''; 
		iStepSet := 5;
	END_IF
(*============================================================================================*)	
5:	sStateReset := 'Sende Service Befehl';
	
	fbStringConvService(
		I_diID:= 			I_stInput.diID,
		I_bServiceOn:= 		bService, 
		I_sStartZeichen:= 	sStartZeichen, 
		I_sEndZeichen:= 	sEndZeichen, 
		Q_sConvString=> 	sSendString);
	
	(* Senden an FiFo*)
	IF GVL_RS485FiFoSend.bSendDoneFiFo[I_FifoID]
	THEN
		sFiFoSend :=	sSendString;
	END_IF
	IF NOT GVL_RS485FiFoSend.bSendDoneFiFo[I_FifoID]
	THEN
		iStepSet := iStepSet+1;
	END_IF
	
(*============================================================================================*)	
6:	sStateReset := 'Sende Service Befehl';

	IF GVL_RS485FiFoSend.bSendDoneFiFo[I_FifoID]
	THEN
		sFiFoSend := ''; 
		iStepSet := 7;
	END_IF
	
(*============================================================================================*)
7:	sStateReset := 'Fertig';
	
	IF bMemWebServer <> bWebServer
		OR bMemWifi <> bWifi
		OR bMemService <> bService 
	THEN
		iStepSet := 0;
	END_IF
	
END_CASE
END_ACTION

ACTION ac02_Ping:
(*============================================================================================*)
(* 	Ping Bautsein, Checkt ob die Kommunikation vorhanden ist *)
(*============================================================================================*)
fbPing(
	I_bExecute:= 			bStartUpCheckPing, 
	I_bAutoPing:= 			bCheckPing, 
	I_bAutoReset:= 			bCheckPing, 
	I_bReset:= 				r_TrigReset.Q
							OR NOT bStartUpCheckPing, 
	I_tPingTimeout:= 		tPingTimer, 
	I_diID:= 				I_stInput.diID, 
	I_sStartZeichen:= 		sStartZeichen, 
	I_sEndZeichen:= 		sEndZeichen, 
	I_StringReceived:= 		I_StringReceived, 
	Q_sState=> , 
	Q_bComOk=> 				bPingOK, 
	Q_bTimeout=> 			bErrorPing);
END_ACTION

ACTION ac10_Counter:
(*============================================================================================*)
(* 	Zähler *)
(*============================================================================================*)
FOR j := 1 TO 6 BY 1 DO 
	r_TrigCountBtn[j](
		CLK := Q_stOutput.bButtons[j]);
		
	IF r_TrigCountBtn[j].Q
	THEN
		Q_stCnt.dwCntButtons[j] := Q_stCnt.dwCntButtons[j]+1;
	END_IF
	
END_FOR
END_ACTION

ACTION ac99_Doku:
(*======================================================================================================================================*)
(*	DOKU	*)
(*======================================================================================================================================*)
(* Wichtiger Hinweis:
		-Bei dem 6 Fach Taster ist zu Beachten, dass es nur 4 Externe EA/s gibt also 4 LEDs und 4 Taster, 
		da der ESP 32 Nur 10Es und 10As besitzt.
		- Die 4 Zusätzlichen Ausgänge werden von der Hintergrundbeleuchtung Ausgeschlossen und müssen über den Befehl: SET_MBR einzeln 
			gesetzt werden! *)	
	
(* Verdrahtung:		
	Verdrahtung füR: KL6041
        +-------+
        |       |
        | TxD+ ----+
        |         |----> RS485 A (zum Bus)
        | RxD+ ----+
        |         |
        | TxD− ----+
        |         |----> RS485 B (zum Bus)
        | RxD− ----+
        +-------+	*)
		
(*======================================================================================================================================*)
(* Telegrammbeschreibung *)

(*	Die XML Dateien der verschiedenen Module sind grundsätzlich immer gleich aufgebaut. 
	Je Instanz der verschiedenen Sensoren und Aktoren werden die zu sendenden Befehle bzw. 
	die zu empfangenen Events beschrieben. 
	Alle Telegramme sind ASCII kodiert und sind umgeben mit dem binären Startzeichen 0xFD und dem binären Endezeichen 0xFE.

	Grundaufbauer aller im Folgenden beschriebenen Telegramme:
	
	-Startzeichen immer 0xFD.
	-Punkte dienen als Trennzeichen der verschiedenen Elemente
	-Endezeichen immer 0xFE.
	-Element 1 ist die Geräte-ID, die entsprechend der verwendeten Module angepasst werden muss (hier beispielhaft jeweils 12345)
	-Element 2 ist ein Schlüsselwort für den jeweiligen Funktionstyp (z.b. BTN, LED, DIM, usw)
	-Element 3 ist die InstanzID gemäß XML Templates (also welche Taster oder welcher Dimmer konkret gemeint ist)
	-Element 4 zeigt die jeweilige Aktion zum Funktionstypen (z.b. ON, OFF, STATUS)
	-Anschließend kommen optional diverse Parameter, die mit P1,P2,...P3 bezeichnet werden
	
	Im Folgenden wird nur noch auf die speziellen Telegramdaten eingegangen:
	
	(*------------------------------------------------------------*)
	Taster oder digitaler Eingang (Sensor):
	(*------------------------------------------------------------*)
	Telegram Event:  	
	
	\xFD 12345.BTN.17.STATUS.P1 \xFE
	
		Funktionstyp:		BTN (kurz für Button)
		Instanz-ID:			hier 17 (in XML nachschauen)
		Aktion:				STATUS
		P1:					1, wenn Taste gedrückt bzw. Eingang aktiv
							0, wenn Taste losgelassen bzw. Eingang inaktiv
	
	Telegram Statusabfrage:  	
	
	\xFD 12345.BTN.17.gSTATUS \xFE
	
		Antwort:  			\xFD 12345.BTN.17.rSTATUS.P1 \xFE
		P1:					1, wenn Taste gedrückt bzw. Eingang aktiv
							0, wenn Taste losgelassen bzw. Eingang inaktiv

	(*------------------------------------------------------------*)
	Led (Aktor):
	(*------------------------------------------------------------*)
	Telegram Helligkeit setzen:  	
	
	\xFD 12345.LED.50.ON.P1.P2.P3 \xFE
	
		Funktionstyp:			LED
		Instanz-ID:				hier 50 (in XML nachschauen)
		Aktion:					ON
		P1:						gewünschte Helligkeit 0-100
		P2:						Einschaltdauer in 100stel Sekunden (0 = daueran)
		P3:						Einschaltverzögerung in Sekunden (0 = ohne Verzögerung)
	
	Telegram Mindesthelligkeit:  	
	
	\xFD 12345.LED.50.SET_MBR.P1 \xFE
		
		Aktion:					SET_MBR (Setzt eine Mindesthelligkeit, die auch dann erhalten bleibt, wenn man per OFF ausschaltet)
		P1:						gewünschte Helligkeit 0-100
	
	Telegram Statusabfrage:  	

	\xFD 12345.LED.50.gSTATUS \xFE
	
		Antwort:  				\xFD 12345.LED.50.rSTATUS.P1.P2 \xFE
		P1:						aktuelle Helligkeit 0-100
		P2:						Einschaltdauer in 100stel Sekunden
	
	(*------------------------------------------------------------*)
	Hintergrundbeleuchtung (Aktor):
	(*------------------------------------------------------------*)
	Telegram Minhelligkeit:  
	
	\xFD 12345.LBN.16.SET_MBR.P1 \xFE
	
		Aktion:					SET_MBR ((Setzt eine Mindesthelligkeit, die auch dann erhalten bleibt, wenn man per OFF ausschaltet)
		P1:						gewünschte Helligkeit 0-100
		
	Telegram Statusabfrage:  	

	\xFD 12345.LBN.16.gSTATUS \xFE
	
		Antwort:  				\xFD 12345.LBN.16.rSTATUS.P1 \xFE
		P1:						aktuelle Helligkeit 0-100

	(*------------------------------------------------------------*)
	Temperatursensor (Sensor):
	(*------------------------------------------------------------*)
	Telegram Event:  	
	
	\xFD 12345.TMP.1.STATUS.P1.P2 \xFE
	
		Funktionstyp:			TMP (kurz für Temperatur)
		Instanz-ID:				hier 1 (in XML nachschauen)
		Aktion:					STATUS
		P1:						Temperatur in Grad Vorkommastellen
		P2:						Temperatur in Grad Nachkommastellen
	
	Telegram Statusabfrage:  
	
	\xFD 12345.TMP.1.gSTATUS \xFE
	
		Antwort:  				\xFD 12345.TMP.1.rSTATUS.P1.P2 \xFE
		P1:						Temperatur in Grad Vorkommastellen
		P2:						Temperatur in Grad Nachkommastellen

	(*------------------------------------------------------------*)
	Feuchtesensor (Sensor):
	(*------------------------------------------------------------*)
	Telegram Event:  	

	\xFD 12345.RHD.1.STATUS.P1.P2 \xFE
	
		Funktionstyp:			RHD (kurz für Relative Humidity)
		Instanz-ID:				hier 1 (in XML nachschauen)
		Aktion:					STATUS
		P1:						Relative Luftfeuchtigkeit 0-100 Vorkommastellen
		P2:						Relative Luftfeuchtigkeit 0-100 Nachkommastellen

	Telegram Statusabfrage:  	
	
	\xFD 12345.RHD.1.gSTATUS \xFE
	
	Antwort:  					\xFD 12345.RHD.1.rSTATUS.P1 \xFE
	P1:							Relative Luftfeuchtigkeit 0-100 Vorkommastellen
	P2:							Relative Luftfeuchtigkeit 0-100 Nachkommastellen

	(*------------------------------------------------------------*)
	Helligkeitssensor (Sensor):
	(*------------------------------------------------------------*)
	Telegram Event:  	
	
	\xFD 12345.BRS.23.STATUS.P1.P2 \xFE
	
		Funktionstyp:			BRS (kurz für Brightness Sensor)
		Instanz-ID:				hier 23 (in XML nachschauen)
		Aktion:					STATUS
		P1:						Relative Helligkeit 0-255 Vorkommastellen
		P2:						Relative Helligkeit 0-255 Nachkommastellen
	
	Telegram Statusabfrage:  	
	
	\xFD 12345.BRS.23.gSTATUS \xFE
	
	Antwort:  					\xFD 12345.BRS.23.rSTATUS.P1 \xFE
	P1:							Relative Helligkeit 0-255 Vorkommastellen
	P2:							Relative Helligkeit 0-255 Nachkommastellen

(*======================================================================================================================================*)
(* Alle Telegramme im Überblick *)	

	<?xml version="1.0" encoding="utf-8"?>
	<Comm Title="Haus-Bus ID 12345" Comment="" Baudrate="57600" Databits="8" Parity="1" EndChar="510">
	<CommCmd Title="6-fach Taster 12345 - Hintergrundbeleuchtung" Comment="" CmdOn="\xFD12345.LBN.16.SET_MBR.&lt;v&gt;.0\xFE" CmdOff="\xFD12345.LBN.16.SET_MBR.0\xFE" Unit="" Analog="true" Text="false" Sensor="false" SourceValHigh="100" DestValHigh="100"/>
	<CommCmd Title="6-fach Taster 12345 - Temperatursensor" Comment="" CmdOn="\xFD12345.TMP.1.STATUS.\v\xFE" CmdOff="" Unit="&lt;v.2&gt;" Analog="true" Text="false" Sensor="true" SourceValHigh="100" DestValHigh="100"/>
	<CommCmd Title="6-fach Taster 12345 - Feuchtesensor" Comment="" CmdOn="\xFD12345.RHD.1.STATUS.\v\xFE" CmdOff="" Unit="&lt;v.x&gt;" Analog="true" Text="false" Sensor="true" SourceValHigh="100" DestValHigh="100"/>
	<CommCmd Title="6-fach Taster 12345 - Helligkeitssensor" Comment="" CmdOn="\xFD12345.BRS.1.STATUS.\v\xFE" CmdOff="" Unit="&lt;v.x&gt;" Analog="true" Text="false" Sensor="true" SourceValHigh="100" DestValHigh="100"/>
	<CommCmd Title="6-fach Taster 12345 - Led 1" Comment="" CmdOn="\xFD12345.LED.49.ON.&lt;v&gt;.0\xFE" CmdOff="\xFD12345.LED.49.OFF\xFE" Unit="" Analog="true" Text="false" Sensor="false" SourceValHigh="100" DestValHigh="100"/>
	<CommCmd Title="6-fach Taster 12345 - Led 2" Comment="" CmdOn="\xFD12345.LED.50.ON.&lt;v&gt;.0\xFE" CmdOff="\xFD12345.LED.50.OFF\xFE" Unit="" Analog="true" Text="false" Sensor="false" SourceValHigh="100" DestValHigh="100"/>
	<CommCmd Title="6-fach Taster 12345 - Led 3" Comment="" CmdOn="\xFD12345.LED.51.ON.&lt;v&gt;.0\xFE" CmdOff="\xFD12345.LED.51.OFF\xFE" Unit="" Analog="true" Text="false" Sensor="false" SourceValHigh="100" DestValHigh="100"/>
	<CommCmd Title="6-fach Taster 12345 - Led 4" Comment="" CmdOn="\xFD12345.LED.52.ON.&lt;v&gt;.0\xFE" CmdOff="\xFD12345.LED.52.OFF\xFE" Unit="" Analog="true" Text="false" Sensor="false" SourceValHigh="100" DestValHigh="100"/>
	<CommCmd Title="6-fach Taster 12345 - Led 5" Comment="" CmdOn="\xFD12345.LED.53.ON.&lt;v&gt;.0\xFE" CmdOff="\xFD12345.LED.53.OFF\xFE" Unit="" Analog="true" Text="false" Sensor="false" SourceValHigh="100" DestValHigh="100"/>
	<CommCmd Title="6-fach Taster 12345 - Led 6" Comment="" CmdOn="\xFD12345.LED.54.ON.&lt;v&gt;.0\xFE" CmdOff="\xFD12345.LED.54.OFF\xFE" Unit="" Analog="true" Text="false" Sensor="false" SourceValHigh="100" DestValHigh="100"/>
	<CommCmd Title="6-fach Taster 12345 - Taster 1" Comment="" CmdOn="\xFD12345.BTN.17.STATUS.\v\xFE" CmdOff="" Unit="&lt;v.x&gt;" Analog="true" Text="false" Sensor="true" SourceValHigh="100" DestValHigh="100"/>
	<CommCmd Title="6-fach Taster 12345 - Taster 2" Comment="" CmdOn="\xFD12345.BTN.18.STATUS.\v\xFE" CmdOff="" Unit="&lt;v.x&gt;" Analog="true" Text="false" Sensor="true" SourceValHigh="100" DestValHigh="100"/>
	<CommCmd Title="6-fach Taster 12345 - Taster 3" Comment="" CmdOn="\xFD12345.BTN.19.STATUS.\v\xFE" CmdOff="" Unit="&lt;v.x&gt;" Analog="true" Text="false" Sensor="true" SourceValHigh="100" DestValHigh="100"/>
	<CommCmd Title="6-fach Taster 12345 - Taster 4" Comment="" CmdOn="\xFD12345.BTN.20.STATUS.\v\xFE" CmdOff="" Unit="&lt;v.x&gt;" Analog="true" Text="false" Sensor="true" SourceValHigh="100" DestValHigh="100"/>
	<CommCmd Title="6-fach Taster 12345 - Taster 5" Comment="" CmdOn="\xFD12345.BTN.21.STATUS.\v\xFE" CmdOff="" Unit="&lt;v.x&gt;" Analog="true" Text="false" Sensor="true" SourceValHigh="100" DestValHigh="100"/>
	<CommCmd Title="6-fach Taster 12345 - Taster 6" Comment="" CmdOn="\xFD12345.BTN.22.STATUS.\v\xFE" CmdOff="" Unit="&lt;v.x&gt;" Analog="true" Text="false" Sensor="true" SourceValHigh="100" DestValHigh="100"/>
	<CommCmd Title="6-fach Taster 12345 - Extern Taster 1" Comment="" CmdOn="\xFD12345.BTN.33.STATUS.\v\xFE" CmdOff="" Unit="&lt;v.x&gt;" Analog="true" Text="false" Sensor="true" SourceValHigh="100" DestValHigh="100"/>
	<CommCmd Title="6-fach Taster 12345 - Extern Taster 2" Comment="" CmdOn="\xFD12345.BTN.34.STATUS.\v\xFE" CmdOff="" Unit="&lt;v.x&gt;" Analog="true" Text="false" Sensor="true" SourceValHigh="100" DestValHigh="100"/>
	<CommCmd Title="6-fach Taster 12345 - Extern Taster 3" Comment="" CmdOn="\xFD12345.BTN.35.STATUS.\v\xFE" CmdOff="" Unit="&lt;v.x&gt;" Analog="true" Text="false" Sensor="true" SourceValHigh="100" DestValHigh="100"/>
	<CommCmd Title="6-fach Taster 12345 - Extern Taster 4" Comment="" CmdOn="\xFD12345.BTN.36.STATUS.\v\xFE" CmdOff="" Unit="&lt;v.x&gt;" Analog="true" Text="false" Sensor="true" SourceValHigh="100" DestValHigh="100"/>
	<CommCmd Title="6-fach Taster 12345 - Extern Taster 5" Comment="" CmdOn="\xFD12345.BTN.37.STATUS.\v\xFE" CmdOff="" Unit="&lt;v.x&gt;" Analog="true" Text="false" Sensor="true" SourceValHigh="100" DestValHigh="100"/>
	<CommCmd Title="6-fach Taster 12345 - Extern Taster 6" Comment="" CmdOn="\xFD12345.BTN.38.STATUS.\v\xFE" CmdOff="" Unit="&lt;v.x&gt;" Analog="true" Text="false" Sensor="true" SourceValHigh="100" DestValHigh="100"/>
	<CommCmd Title="6-fach Taster 12345 - Extern Led 1" Comment="" CmdOn="\xFD12345.LED.65.ON.&lt;v&gt;.0\xFE" CmdOff="\xFD12345.LED.65.OFF\xFE" Unit="" Analog="true" Text="false" Sensor="false" SourceValHigh="100" DestValHigh="100"/>
	<CommCmd Title="6-fach Taster 12345 - Extern Led 2" Comment="" CmdOn="\xFD12345.LED.66.ON.&lt;v&gt;.0\xFE" CmdOff="\xFD12345.LED.66.OFF\xFE" Unit="" Analog="true" Text="false" Sensor="false" SourceValHigh="100" DestValHigh="100"/>
	<CommCmd Title="6-fach Taster 12345 - Extern Led 3" Comment="" CmdOn="\xFD12345.LED.67.ON.&lt;v&gt;.0\xFE" CmdOff="\xFD12345.LED.67.OFF\xFE" Unit="" Analog="true" Text="false" Sensor="false" SourceValHigh="100" DestValHigh="100"/>
	<CommCmd Title="6-fach Taster 12345 - Extern Led 4" Comment="" CmdOn="\xFD12345.LED.68.ON.&lt;v&gt;.0\xFE" CmdOff="\xFD12345.LED.68.OFF\xFE" Unit="" Analog="true" Text="false" Sensor="false" SourceValHigh="100" DestValHigh="100"/>
	<CommCmd Title="6-fach Taster 12345 - Extern Led 5" Comment="" CmdOn="\xFD12345.LED.69.ON.&lt;v&gt;.0\xFE" CmdOff="\xFD12345.LED.69.OFF\xFE" Unit="" Analog="true" Text="false" Sensor="false" SourceValHigh="100" DestValHigh="100"/>
	<CommCmd Title="6-fach Taster 12345 - Extern Led 6" Comment="" CmdOn="\xFD12345.LED.70.ON.&lt;v&gt;.0\xFE" CmdOff="\xFD12345.LED.70.OFF\xFE" Unit="" Analog="true" Text="false" Sensor="false" SourceValHigh="100" DestValHigh="100"/>
	<CommCmd Title="6-fach Taster 12345 - RFID Leser" Comment="" CmdOn="\xFD12345.RFD.65.TAG_ID.\v\xFE" CmdOff="" Unit="&lt;v.x&gt;" Analog="false" Text="true" Sensor="true" SourceValHigh="100" DestValHigh="100"/>
	<CommCmd Title="6-fach Taster 12345 - RFID Leser" Comment="" CmdOn="\xFD12345.RFD.66.TAG_ID.\v\xFE" CmdOff="" Unit="&lt;v.x&gt;" Analog="false" Text="true" Sensor="true" SourceValHigh="100" DestValHigh="100"/>
	<CommCmd Title="6-fach Taster 12345 - RFID Leser" Comment="" CmdOn="\xFD12345.RFD.67.TAG_ID.\v\xFE" CmdOff="" Unit="&lt;v.x&gt;" Analog="false" Text="true" Sensor="true" SourceValHigh="100" DestValHigh="100"/>
	<CommCmd Title="6-fach Taster 12345 - RFID Leser" Comment="" CmdOn="\xFD12345.RFD.68.TAG_ID.\v\xFE" CmdOff="" Unit="&lt;v.x&gt;" Analog="false" Text="true" Sensor="true" SourceValHigh="100" DestValHigh="100"/>
	<CommCmd Title="6-fach Taster 12345 - RFID Leser" Comment="" CmdOn="\xFD12345.RFD.69.TAG_ID.\v\xFE" CmdOff="" Unit="&lt;v.x&gt;" Analog="false" Text="true" Sensor="true" SourceValHigh="100" DestValHigh="100"/>
	</Comm>
*)
END_ACTION

END_FUNCTION_BLOCK

// ---- POUs/RS485_Hausbus_FB/CYD/fb_StringConvCYDWeb.TcPOU
(*======================================================================================================================================*)
(*fb_StringConvTB6F:	Zusammensetzen des Strings für 6Fach Bust Taster (LEDs und Hintergrundbeleuchtung und Reset)*)
(*
Date          	| Version    	| created under        	| Author          	| Remark *)
(*====================================================================================================================================================*)
(*05/05/2025   	| 1.00      		| TC3		  		| N.Kersting       | first release *)
(*06/05/2025   	| 1.01      		| TC3		  		| N.Kersting       | Externe LEDs Nachgerüstet *)
(*08/05/2025   	| 1.02      		| TC3		  		| N.Kersting       | Umschaltung ob Externe LEDs verwendet werden oder nicht *)
(*22/05/2025   	| 1.03      		| TC3		  		| N.Kersting       | Spezialversion für CYD *)
(*====================================================================================================================================================*)
FUNCTION_BLOCK fb_StringConvCYDWeb
VAR_INPUT
	I_diID				:DINT;							(* Device ID *)
	I_bWebOn			:BOOL;
	I_sStartZeichen		:BYTE := 16#FD;					(* Startzeichen Präfix *)
	I_sEndZeichen		:BYTE := 16#FE;					(* Endzeichen Suffix *)
END_VAR
VAR_OUTPUT
	Q_sConvString		:STRING(255);
END_VAR
VAR
END_VAR


